           1200:
               gtyp_VGR.Workpiece.s_id := '0';
               gtyp_VGR.Workpiece.s_state := '';
               gtyp_VGR.Workpiece.s_type := '';
               FOR li_Counter := 1 TO 8 DO
                   gtyp_VGR.History[li_Counter].i_code := 0;
                   gtyp_VGR.History[li_Counter].ldt_ts := DT#1990-01-01-00:00:00.00;
               END_FOR;

               IF gtyp_HBW.x_HBW_Container_Available THEN
                   gtyp_VGR.x_HBW_Discards := TRUE;
               END_IF;

               IF gtyp_HBW.x_HBW_Discards_Accepted OR gtyp_HBW.x_HBW_PickedUp_Accepted THEN
                   gtyp_VGR.x_HBW_Discards := FALSE;
                   gtyp_VGR.x_HBW_PickedUp := FALSE;
                   gtyp_HBW.x_HBW_Discards_Accepted := FALSE;
                   gtyp_HBW.x_HBW_PickedUp_Accepted := FALSE;
               END_IF;

               li_Lights := 2;
               gtyp_VGR.vertical_Axis.x_Reference := TRUE;

               IF NOT gtyp_VGR.vertical_Axis.x_Referenced THEN
                   li_StepCase := 1210;
               END_IF;

           1210:
               IF gtyp_VGR.vertical_Axis.x_Referenced THEN
                   gtyp_VGR.vertical_Axis.x_Reference := FALSE;
                   li_StepCase := 1220;
               END_IF;

           1220:
               gtyp_VGR.horizontal_Axis.x_Reference := TRUE;

               IF NOT gtyp_VGR.horizontal_Axis.x_Referenced THEN
                   li_StepCase := 1230;
               END_IF;

           1230:
               IF gtyp_VGR.horizontal_Axis.x_Referenced THEN
                   gtyp_VGR.horizontal_Axis.x_Reference := FALSE;
                   li_StepCase := 1240;
               END_IF;

           1240:
               gtyp_VGR.rotate_Axis.x_Reference := TRUE;

               IF NOT gtyp_VGR.rotate_Axis.x_Referenced THEN
                   li_StepCase := 1250;
               END_IF;

           1250:
               IF gtyp_VGR.rotate_Axis.x_Referenced THEN
                   gtyp_VGR.rotate_Axis.x_Reference := FALSE;
                   li_StepCase := 1260;
               END_IF;

           1260:
               gtyp_VGR.horizontal_Axis.di_Target_Position := gtyp_VGR.di_Pos_NiO_horizontal;
               gtyp_VGR.horizontal_Axis.x_Start_Positioning := TRUE;
               gtyp_VGR.vertical_Axis.di_Target_Position := gtyp_VGR.di_Pos_NiO_vertical;
               gtyp_VGR.vertical_Axis.x_Start_Positioning := TRUE;
               gtyp_VGR.vertical_Axis.i_PWM := 500;
               gtyp_VGR.rotate_Axis.di_Target_Position := gtyp_VGR.di_Pos_NiO_rotate;
               gtyp_VGR.rotate_Axis.x_Start_Positioning := TRUE;

               IF (gtyp_VGR.horizontal_Axis.di_Actual_Position <= (gtyp_VGR.di_Pos_NiO_horizontal + gtyp_VGR.horizontal_Axis.Config.di_Pos_Window))
                   AND (gtyp_VGR.horizontal_Axis.di_Actual_Position >= (gtyp_VGR.di_Pos_NiO_horizontal - gtyp_VGR.horizontal_Axis.Config.di_Pos_Window))
                   AND gtyp_VGR.horizontal_Axis.x_Position_Reached THEN
                   gtyp_VGR.horizontal_Axis.x_Start_Positioning := FALSE;
               END_IF;

               IF (gtyp_VGR.vertical_Axis.di_Actual_Position <= (gtyp_VGR.di_Pos_NiO_vertical + gtyp_VGR.vertical_Axis.Config.di_Pos_Window))
                   AND (gtyp_VGR.vertical_Axis.di_Actual_Position >= (gtyp_VGR.di_Pos_NiO_vertical - gtyp_VGR.vertical_Axis.Config.di_Pos_Window))
                   AND gtyp_VGR.vertical_Axis.x_Position_Reached THEN
                   gtyp_VGR.vertical_Axis.x_Start_Positioning := FALSE;
               END_IF;

               IF (gtyp_VGR.rotate_Axis.di_Actual_Position <= (gtyp_VGR.di_Pos_NiO_rotate + gtyp_VGR.rotate_Axis.Config.di_Pos_Window))
                   AND (gtyp_VGR.rotate_Axis.di_Actual_Position >= (gtyp_VGR.di_Pos_NiO_rotate - gtyp_VGR.rotate_Axis.Config.di_Pos_Window))
                   AND gtyp_VGR.rotate_Axis.x_Position_Reached THEN
                   gtyp_VGR.rotate_Axis.x_Start_Positioning := FALSE;
               END_IF;

               IF (gtyp_VGR.horizontal_Axis.di_Actual_Position <= (gtyp_VGR.di_Pos_NiO_horizontal + gtyp_VGR.horizontal_Axis.Config.di_Pos_Window))
                   AND (gtyp_VGR.horizontal_Axis.di_Actual_Position >= (gtyp_VGR.di_Pos_NiO_horizontal - gtyp_VGR.horizontal_Axis.Config.di_Pos_Window))
                   AND gtyp_VGR.horizontal_Axis.x_Position_Reached
                   AND (gtyp_VGR.vertical_Axis.di_Actual_Position <= (gtyp_VGR.di_Pos_NiO_vertical + gtyp_VGR.vertical_Axis.Config.di_Pos_Window))
                   AND (gtyp_VGR.vertical_Axis.di_Actual_Position >= (gtyp_VGR.di_Pos_NiO_vertical - gtyp_VGR.vertical_Axis.Config.di_Pos_Window))
                   AND gtyp_VGR.vertical_Axis.x_Position_Reached
                   AND (gtyp_VGR.rotate_Axis.di_Actual_Position <= (gtyp_VGR.di_Pos_NiO_rotate + gtyp_VGR.rotate_Axis.Config.di_Pos_Window))
                   AND (gtyp_VGR.rotate_Axis.di_Actual_Position >= (gtyp_VGR.di_Pos_NiO_rotate - gtyp_VGR.rotate_Axis.Config.di_Pos_Window))
                   AND gtyp_VGR.rotate_Axis.x_Position_Reached THEN
                   gtyp_VGR.horizontal_Axis.x_Start_Positioning := FALSE;
                   gtyp_VGR.vertical_Axis.x_Start_Positioning := FALSE;
                   gtyp_VGR.rotate_Axis.x_Start_Positioning := FALSE;
                   gtyp_VGR.vertical_Axis.i_PWM := 800;
                   li_StepCase := 1270;
               END_IF;

           1270:
               QX_VGR_ValveVacuum_Q8 := FALSE;
               li_StepCase := 1280;

           1280:

               lx_Start_TON_Wait := TRUE;
               lt_TON_Wait := T#1000ms;

               IF lfb_TON_Wait.Q THEN
                   QX_VGR_Compressor_Q7  := FALSE;
                   lx_Start_TON_Wait               := FALSE;
                   gtyp_VGR.x_Workpiece_NiO := FALSE;
                   gtyp_VGR.x_HBW_Discards := FALSE;
                   li_Lights := 1;
                   li_StepCase            := 0;
               END_IF;

       ELSE
               ;
       END_CASE;

   ELSE
       gtyp_VGR.Workpiece.s_id := '';
       gtyp_VGR.Workpiece.s_state := '';
       gtyp_VGR.Workpiece.s_type := '';

       gtyp_VGR.x_State_Process := FALSE;
       gtyp_Interface_Dashboard.Subscribe.State_Order.ldt_ts := DT_TO_LDT(ldt_MQTT);
       gtyp_Interface_Dashboard.Subscribe.State_Order.s_state := 'WAITING_FOR_ORDER';
       gtyp_Interface_Dashboard.Subscribe.State_Order.s_type := '';
       FOR li_Counter := 1 TO 8 DO
           gtyp_VGR.History[li_Counter].i_code := 0;
           gtyp_VGR.History[li_Counter].ldt_ts := DT#1990-01-01-00:00:00.00;
       END_FOR;

       gtyp_VGR.x_Start_Park_Position    := FALSE;
       gtyp_VGR.x_Park_Position_Reached  := FALSE;
       gtyp_VGR.x_NFC_Start_First        := FALSE;
       gtyp_VGR.x_NFC_Start              := FALSE;
       gtyp_VGR.x_NFC_Completed          := FALSE;
       gtyp_VGR.x_HBW_Storage            := FALSE;
       gtyp_VGR.x_HBW_Outsource          := FALSE;
       gtyp_VGR.s_HBW_Outsource_Typ      := '';
       gtyp_VGR.x_HBW_Discards           := FALSE;
       gtyp_VGR.x_HBW_PickedUp           := FALSE;
       gtyp_VGR.x_MPO_Req_Discard        := FALSE;
       gtyp_VGR.x_MPO_Discards           := FALSE;
       gtyp_VGR.x_Ready_For_Outsource    := FALSE;
       gtyp_VGR.x_State_Process          := FALSE;
       gtyp_VGR.x_Workpiece_NiO          := FALSE;

       gtyp_VGR.vertical_Axis.i_PWM      := 800;

       li_Lights := 1;
       lx_Init := TRUE;
   END_IF;
END_FUNCTION_BLOCK

FUNCTION_BLOCK PRG_Order
   VAR
      lx_Init : Bool;
      li_StepCase : Int;
      lldt_ts_old : LDT;
      ldt_MQTT : Date_And_Time;
      li_Return_LDT : Int;
      lfb_TON_Wait : TON_TIME;
      lx_Start_TON_Wait : Bool;
   END_VAR

   IF lx_Init THEN
       lfb_TON_Wait(IN:= lx_Start_TON_Wait,PT:= T#20s);
       CASE li_StepCase OF

           0:
               lx_Start_TON_Wait := FALSE;
               li_StepCase := 10;

           10:
               IF (gtyp_Interface_Dashboard.Publish.OrderWorkpieceButton.ldt_ts > lldt_ts_old) THEN
                   li_Return_LDT := RD_SYS_T(ldt_MQTT);
                   gtyp_Interface_Dashboard.Subscribe.State_Order.ldt_ts := DT_TO_LDT(ldt_MQTT);
                   gtyp_Interface_Dashboard.Subscribe.State_Order.s_state := 'ORDERED';
                   gtyp_VGR.s_HBW_Outsource_Typ := gtyp_Interface_Dashboard.Publish.OrderWorkpieceButton.s_type;
                   gtyp_Interface_Dashboard.Subscribe.State_Order.s_type := gtyp_VGR.s_HBW_Outsource_Typ;
                   IF gtyp_VGR.x_Ready_For_Outsource THEN
                       lldt_ts_old := gtyp_Interface_Dashboard.Publish.OrderWorkpieceButton.ldt_ts;
                       gtyp_VGR.x_HBW_Outsource := TRUE;
                       li_StepCase := 20;
                   END_IF;
               END_IF;

           20:
               IF gtyp_VGR.x_HBW_PickedUp OR NOT gtyp_VGR.x_HBW_Outsource THEN
                   gtyp_VGR.x_HBW_Outsource := FALSE;
                   gtyp_VGR.s_HBW_Outsource_Typ := '';
                   li_StepCase := 0;
               END_IF;


       ELSE
                   ;
       END_CASE;

   ELSE
       lx_Init    := TRUE;
       lldt_ts_old:= DT#1970-01-01-00:00:00.00;
   END_IF;
END_FUNCTION_BLOCK

FUNCTION_BLOCK PRG_MPO_Set_Park_Position
   VAR
      lx_Init : Bool;
      lx_Start_TON_Wait : Bool;
      lt_TON_Wait : Time;
      li_StepCase : Int;
      lfb_TON_Wait : TON_TIME;
      lfb_R_Trig_Start_Park_Pos : R_TRIG;
   END_VAR



   IF lx_Init THEN


       lfb_TON_Wait(IN := lx_Start_TON_Wait,
                     PT := lt_TON_Wait);

       lfb_R_Trig_Start_Park_Pos(CLK := gtyp_Setup.x_Park_Position
                                  OR IX_Set_Park_Position);


       IF lfb_R_Trig_Start_Park_Pos.Q THEN
           gtyp_MPO.x_Start_Park_Position := TRUE;
           li_StepCase := 0;
       END_IF;


       IF NOT gtyp_MPO.x_Start_Park_Position THEN
           li_StepCase := 0;
       END_IF;


       CASE li_StepCase OF

           0:
               lx_Start_TON_Wait := FALSE;
               li_StepCase := 10;

           10:
               IF gtyp_MPO.x_Start_Park_Position AND NOT gtyp_MPO.x_Park_Position_Reached THEN
                   li_StepCase := 20;
               END_IF;

           20:
               QX_MPO_M5_VacuumTowardsTurnTable_Q8 := FALSE;
               QX_MPO_M5_VacuumTowardsOven_Q7    := TRUE;
               lx_Start_TON_Wait                  := TRUE;
               lt_TON_Wait                        := T#4000ms;

               IF lfb_TON_Wait.Q THEN
                   QX_MPO_M5_VacuumTowardsTurnTable_Q8 := FALSE;
                   QX_MPO_M5_VacuumTowardsOven_Q7    := FALSE;
                   lx_Start_TON_Wait                  := FALSE;
                   li_StepCase                        := 30;
               END_IF;

           30:
               QX_MPO_M1_TurnTableClockwise_Q1        := TRUE;
               QX_MPO_M1_TurnTableCounterclockwise_Q2 := FALSE;
               lx_Start_TON_Wait := TRUE;
               lt_TON_Wait := T#1000ms;

               IF lfb_TON_Wait.Q THEN
                   QX_MPO_M1_TurnTableClockwise_Q1 := FALSE;
                   QX_MPO_M1_TurnTableCounterclockwise_Q2 := FALSE;
                   lx_Start_TON_Wait := FALSE;
                   li_StepCase := 40;
               END_IF;

           40:
               gtyp_MPO.x_Park_Position_Reached := TRUE;



           ELSE
               ;
       END_CASE;

   ELSE
       lx_Init := TRUE;
   END_IF;
END_FUNCTION_BLOCK

FUNCTION_BLOCK PRG_HBW_Ablauf
   VAR
      lx_Init : Bool;
      lx_Start_TON_Fill_HBW : Bool;
      lx_Start_TON_Wait : Bool;
      lx_Time_Error : Bool;
      lt_TON_Wait : Time;
      lx_Start_TON_State : Bool;
      lx_Storage : Bool;
      ldt_MQTT : Date_And_Time;
      li_Return_LDT : Int;
      lldt_Outsource : LDT;
      li_Lights : Int;
      li_Lights_old : Int;
      li_Counter_Hor : Int;
      li_Counter_Ver : Int;
      li_Counter_Act_Hor : Int;
      li_Counter_Act_Ver : Int;
      li_Counter : Int;
      li_StepCase : Int;
      ldi_PosRack_Horizontal : DInt;
      ldi_PosRack_Vertical : DInt;
      ls_Color : String;
      lfb_TON_State : TON_TIME;
      lfb_TON_ConveyerBelt_Out : TON_TIME;
      lfb_TON_Wait : TON_TIME;
      lfb_TON_Fill_HBW : TON_TIME;
      lfb_TON_Error : TON_TIME;
   END_VAR

   IF lx_Init THEN
       IF gtyp_Setup.x_Set_Pos_Activ OR gtyp_HBW.x_Start_Park_Position THEN
           li_StepCase := 0;
       END_IF;


       lfb_TON_State(IN := NOT lx_Start_TON_State,
                       PT := T#2s);


       lfb_TON_Error(IN := lx_Time_Error,
                      PT := T#30s);


       lfb_TON_Fill_HBW(IN := lx_Start_TON_Fill_HBW,
                         PT := T#60s);

       IF lfb_TON_Fill_HBW.Q THEN
           lx_Start_TON_Fill_HBW:= FALSE;
       END_IF;

       IF lx_Start_TON_Fill_HBW AND (IX_Fill_HBW OR gtyp_Setup.x_Fill_Rack_HBW) THEN
           li_Return_LDT := RD_SYS_T(ldt_MQTT);

           gtyp_HBW.Rack_Workpiece[1, 1].s_id    := '04c34892186580';
           gtyp_HBW.Rack_Workpiece[1, 1].s_state := 'RAW';
           gtyp_HBW.Rack_Workpiece[1, 1].s_type  := 'WHITE';
           gtyp_HBW.Rack_History[1, 1].History[1].ldt_ts := DT_TO_LDT(ldt_MQTT);
           gtyp_HBW.Rack_History[1, 1].History[1].i_code := 100;
           gtyp_HBW.Rack_History[1, 1].History[2].ldt_ts := DT_TO_LDT(ldt_MQTT);
           gtyp_HBW.Rack_History[1, 1].History[2].i_code := 200;
           gtyp_HBW.Rack_History[1, 1].History[3].ldt_ts := DT_TO_LDT(ldt_MQTT);
           gtyp_HBW.Rack_History[1, 1].History[3].i_code := 300;

           gtyp_HBW.Rack_Workpiece[1, 2].s_id    := '04c34892186581';
           gtyp_HBW.Rack_Workpiece[1, 2].s_state := 'RAW';
           gtyp_HBW.Rack_Workpiece[1, 2].s_type  := 'WHITE';
           gtyp_HBW.Rack_History[1, 2].History[1].ldt_ts := DT_TO_LDT(ldt_MQTT);
           gtyp_HBW.Rack_History[1, 2].History[1].i_code := 100;
           gtyp_HBW.Rack_History[1, 2].History[2].ldt_ts := DT_TO_LDT(ldt_MQTT);
           gtyp_HBW.Rack_History[1, 2].History[2].i_code := 200;
           gtyp_HBW.Rack_History[1, 2].History[3].ldt_ts := DT_TO_LDT(ldt_MQTT);
           gtyp_HBW.Rack_History[1, 2].History[3].i_code := 300;

           gtyp_HBW.Rack_Workpiece[1, 3].s_id    := '04c34892186582';
           gtyp_HBW.Rack_Workpiece[1, 3].s_state := 'RAW';
           gtyp_HBW.Rack_Workpiece[1, 3].s_type  := 'WHITE';
           gtyp_HBW.Rack_History[1, 3].History[1].ldt_ts := DT_TO_LDT(ldt_MQTT);
           gtyp_HBW.Rack_History[1, 3].History[1].i_code := 100;
           gtyp_HBW.Rack_History[1, 3].History[2].ldt_ts := DT_TO_LDT(ldt_MQTT);
           gtyp_HBW.Rack_History[1, 3].History[2].i_code := 200;
           gtyp_HBW.Rack_History[1, 3].History[3].ldt_ts := DT_TO_LDT(ldt_MQTT);
           gtyp_HBW.Rack_History[1, 3].History[3].i_code := 300;

           gtyp_HBW.Rack_Workpiece[2, 1].s_id    := '04c34892186583';
           gtyp_HBW.Rack_Workpiece[2, 1].s_state := 'RAW';
           gtyp_HBW.Rack_Workpiece[2, 1].s_type  := 'RED';
           gtyp_HBW.Rack_History[2, 1].History[1].ldt_ts := DT_TO_LDT(ldt_MQTT);
           gtyp_HBW.Rack_History[2, 1].History[1].i_code := 100;
           gtyp_HBW.Rack_History[2, 1].History[2].ldt_ts := DT_TO_LDT(ldt_MQTT);
           gtyp_HBW.Rack_History[2, 1].History[2].i_code := 200;
           gtyp_HBW.Rack_History[2, 1].History[3].ldt_ts := DT_TO_LDT(ldt_MQTT);
           gtyp_HBW.Rack_History[2, 1].History[3].i_code := 300;

           gtyp_HBW.Rack_Workpiece[2, 2].s_id    := '04c34892186584';
           gtyp_HBW.Rack_Workpiece[2, 2].s_state := 'RAW';
           gtyp_HBW.Rack_Workpiece[2, 2].s_type  := 'RED';
           gtyp_HBW.Rack_History[2, 2].History[1].ldt_ts := DT_TO_LDT(ldt_MQTT);
           gtyp_HBW.Rack_History[2, 2].History[1].i_code := 100;
           gtyp_HBW.Rack_History[2, 2].History[2].ldt_ts := DT_TO_LDT(ldt_MQTT);
           gtyp_HBW.Rack_History[2, 2].History[2].i_code := 200;
           gtyp_HBW.Rack_History[2, 2].History[3].ldt_ts := DT_TO_LDT(ldt_MQTT);
           gtyp_HBW.Rack_History[2, 2].History[3].i_code := 300;

           gtyp_HBW.Rack_Workpiece[2, 3].s_id    := '04c34892186585';
           gtyp_HBW.Rack_Workpiece[2, 3].s_state := 'RAW';
           gtyp_HBW.Rack_Workpiece[2, 3].s_type  := 'RED';
           gtyp_HBW.Rack_History[2, 3].History[1].ldt_ts := DT_TO_LDT(ldt_MQTT);
           gtyp_HBW.Rack_History[2, 3].History[1].i_code := 100;
           gtyp_HBW.Rack_History[2, 3].History[2].ldt_ts := DT_TO_LDT(ldt_MQTT);
           gtyp_HBW.Rack_History[2, 3].History[2].i_code := 200;
           gtyp_HBW.Rack_History[2, 3].History[3].ldt_ts := DT_TO_LDT(ldt_MQTT);
           gtyp_HBW.Rack_History[2, 3].History[3].i_code := 300;

           gtyp_HBW.Rack_Workpiece[3, 1].s_id    := '04c34892186586';
           gtyp_HBW.Rack_Workpiece[3, 1].s_state := 'RAW';
           gtyp_HBW.Rack_Workpiece[3, 1].s_type  := 'BLUE';
           gtyp_HBW.Rack_History[3, 1].History[1].ldt_ts := DT_TO_LDT(ldt_MQTT);
           gtyp_HBW.Rack_History[3, 1].History[1].i_code := 100;
           gtyp_HBW.Rack_History[3, 1].History[2].ldt_ts := DT_TO_LDT(ldt_MQTT);
           gtyp_HBW.Rack_History[3, 1].History[2].i_code := 200;
           gtyp_HBW.Rack_History[3, 1].History[3].ldt_ts := DT_TO_LDT(ldt_MQTT);
           gtyp_HBW.Rack_History[3, 1].History[3].i_code := 300;

           gtyp_HBW.Rack_Workpiece[3, 2].s_id    := '04c34892186587';
           gtyp_HBW.Rack_Workpiece[3, 2].s_state := 'RAW';
           gtyp_HBW.Rack_Workpiece[3, 2].s_type  := 'BLUE';
           gtyp_HBW.Rack_History[3, 2].History[1].ldt_ts := DT_TO_LDT(ldt_MQTT);
           gtyp_HBW.Rack_History[3, 2].History[1].i_code := 100;
           gtyp_HBW.Rack_History[3, 2].History[2].ldt_ts := DT_TO_LDT(ldt_MQTT);
           gtyp_HBW.Rack_History[3, 2].History[2].i_code := 200;
           gtyp_HBW.Rack_History[3, 2].History[3].ldt_ts := DT_TO_LDT(ldt_MQTT);
           gtyp_HBW.Rack_History[3, 2].History[3].i_code := 300;

           gtyp_HBW.Rack_Workpiece[3, 3].s_id    := '04c34892186588';
           gtyp_HBW.Rack_Workpiece[3, 3].s_state := 'RAW';
           gtyp_HBW.Rack_Workpiece[3, 3].s_type  := 'BLUE';
           gtyp_HBW.Rack_History[3, 3].History[1].ldt_ts := DT_TO_LDT(ldt_MQTT);
           gtyp_HBW.Rack_History[3, 3].History[1].i_code := 100;
           gtyp_HBW.Rack_History[3, 3].History[2].ldt_ts := DT_TO_LDT(ldt_MQTT);
           gtyp_HBW.Rack_History[3, 3].History[2].i_code := 200;
           gtyp_HBW.Rack_History[3, 3].History[3].ldt_ts := DT_TO_LDT(ldt_MQTT);
           gtyp_HBW.Rack_History[3, 3].History[3].i_code := 300;

           lx_Start_TON_Fill_HBW          := FALSE;
           gtyp_Setup.x_Fill_Rack_HBW    := FALSE;
       END_IF;

       gtyp_Setup.x_Start_TON_Fill_HBW := lx_Start_TON_Fill_HBW;


        IF (lfb_TON_State.Q OR (li_Lights <> li_Lights_old)) AND NOT lx_Start_TON_State THEN
           li_Lights_old := li_Lights;
           lx_Start_TON_State := TRUE;
           li_Return_LDT := RD_SYS_T(ldt_MQTT);
           gtyp_Interface_Dashboard.Subscribe.Stock_HBW.StockItem := gtyp_HBW.Rack_Workpiece;
           gtyp_Interface_Dashboard.Subscribe.Stock_HBW.ldt_ts := DT_TO_LDT(ldt_MQTT);

           gtyp_Interface_Dashboard.Subscribe.State_HBW.ldt_ts := DT_TO_LDT(ldt_MQTT);
           gtyp_Interface_Dashboard.Subscribe.State_HBW.i_code := li_Lights;
           gtyp_Interface_Dashboard.Subscribe.State_HBW.s_description := '';
           gtyp_Interface_Dashboard.Subscribe.State_HBW.s_station := 'hbw';
           gtyp_Interface_Dashboard.Subscribe.State_HBW.s_target := '';
       END_IF;


       IF NOT lfb_TON_State.Q AND lx_Start_TON_State THEN
           lx_Start_TON_State := FALSE;
       END_IF;


       lfb_TON_Wait(IN := lx_Start_TON_Wait,
                       PT := lt_TON_Wait);


       lfb_TON_ConveyerBelt_Out(IN := NOT IX_HBW_LightBarrierOutside_I3,
                                 PT := T#300ms);



       gtyp_HBW.Rack_Pos[1, 1].di_PosRack_Horizontal := gtyp_HBW.di_PosRack_A1_Horizontal;
       gtyp_HBW.Rack_Pos[2, 1].di_PosRack_Horizontal := gtyp_HBW.di_PosRack_A1_Horizontal;
       gtyp_HBW.Rack_Pos[3, 1].di_PosRack_Horizontal := gtyp_HBW.di_PosRack_A1_Horizontal;

       gtyp_HBW.Rack_Pos[1, 2].di_PosRack_Horizontal := gtyp_HBW.di_PosRack_B2_Horizontal;
       gtyp_HBW.Rack_Pos[2, 2].di_PosRack_Horizontal := gtyp_HBW.di_PosRack_B2_Horizontal;
       gtyp_HBW.Rack_Pos[3, 2].di_PosRack_Horizontal := gtyp_HBW.di_PosRack_B2_Horizontal;

       gtyp_HBW.Rack_Pos[1, 3].di_PosRack_Horizontal := gtyp_HBW.di_PosRack_C3_Horizontal;
       gtyp_HBW.Rack_Pos[2, 3].di_PosRack_Horizontal := gtyp_HBW.di_PosRack_C3_Horizontal;
       gtyp_HBW.Rack_Pos[3, 3].di_PosRack_Horizontal := gtyp_HBW.di_PosRack_C3_Horizontal;

       gtyp_HBW.Rack_Pos[1, 1].di_PosRack_Vertical := gtyp_HBW.di_PosRack_A1_Vertical;
       gtyp_HBW.Rack_Pos[1, 2].di_PosRack_Vertical := gtyp_HBW.di_PosRack_A1_Vertical;
       gtyp_HBW.Rack_Pos[1, 3].di_PosRack_Vertical := gtyp_HBW.di_PosRack_A1_Vertical;

       gtyp_HBW.Rack_Pos[2, 1].di_PosRack_Vertical := gtyp_HBW.di_PosRack_B2_Vertical;
       gtyp_HBW.Rack_Pos[2, 2].di_PosRack_Vertical := gtyp_HBW.di_PosRack_B2_Vertical;
       gtyp_HBW.Rack_Pos[2, 3].di_PosRack_Vertical := gtyp_HBW.di_PosRack_B2_Vertical;

       gtyp_HBW.Rack_Pos[3, 1].di_PosRack_Vertical := gtyp_HBW.di_PosRack_C3_Vertical;
       gtyp_HBW.Rack_Pos[3, 2].di_PosRack_Vertical := gtyp_HBW.di_PosRack_C3_Vertical;
       gtyp_HBW.Rack_Pos[3, 3].di_PosRack_Vertical := gtyp_HBW.di_PosRack_C3_Vertical;


       CASE li_StepCase OF

           0:
               lx_Start_TON_Wait := FALSE;
               lx_Time_Error := FALSE;

               gtyp_HBW.Horizontal_Axis.x_Start_Positioning := FALSE;
               gtyp_HBW.Vertical_Axis.x_Start_Positioning := FALSE;
               gtyp_HBW.Horizontal_Axis.x_Reference := FALSE;
               gtyp_HBW.Vertical_Axis.x_Reference := FALSE;

               IF NOT gtyp_HBW.x_Error AND NOT gtyp_Setup.x_Set_Pos_Activ AND NOT gtyp_HBW.x_Start_Park_Position THEN
                   li_StepCase := 10;
               END_IF;

           10:
               li_Lights := 2;
               IF IX_HBW_SwitchCantileverFront_I5 OR NOT IX_HBW_SwitchCantileverBack_I6 THEN
                   QX_HBW_M4_CantileverBackward_Q8 := TRUE;
                   QX_HBW_M4_CantileverForward_Q7 := FALSE;
               ELSIF NOT IX_HBW_SwitchCantileverFront_I5 AND IX_HBW_SwitchCantileverBack_I6 THEN
                   QX_HBW_M4_CantileverBackward_Q8 := FALSE;
                   QX_HBW_M4_CantileverForward_Q7 := FALSE;
                   li_StepCase := 20;
               END_IF;

           20:

               gtyp_HBW.Horizontal_Axis.x_Reference := TRUE;
               gtyp_HBW.Vertical_Axis.x_Reference := TRUE;

               IF NOT gtyp_HBW.Horizontal_Axis.x_Referenced AND NOT gtyp_HBW.Vertical_Axis.x_Referenced THEN
                   li_StepCase := 30;
               END_IF;

           30:
               IF gtyp_HBW.Horizontal_Axis.x_Referenced THEN
                   gtyp_HBW.Horizontal_Axis.x_Reference := FALSE;
               END_IF;
               IF gtyp_HBW.Vertical_Axis.x_Referenced THEN
                   gtyp_HBW.Vertical_Axis.x_Reference := FALSE;
               END_IF;

               IF gtyp_HBW.Horizontal_Axis.x_Referenced AND gtyp_HBW.Vertical_Axis.x_Referenced THEN
                   gtyp_HBW.Horizontal_Axis.x_Reference := FALSE;
                   gtyp_HBW.Vertical_Axis.x_Reference := FALSE;
                   li_StepCase := 40;
               END_IF;

           40:

               li_Lights := 1;
               lx_Storage := FALSE;


               IF gtyp_VGR.x_HBW_Storage THEN
                   li_Lights := 2;
                   li_StepCase := 50;

               ELSIF gtyp_VGR.x_HBW_Outsource THEN
                   li_Lights := 2;
                   li_StepCase := 60;
               END_IF;

           50:
               FOR li_Counter_Hor := 1 TO 3 DO
                   FOR li_Counter_Ver := 1 TO 3 DO
                       IF gtyp_HBW.Rack_Workpiece[li_Counter_Ver, li_Counter_Hor].s_id = '0' THEN
                           li_Counter_Act_Hor := li_Counter_Hor;
                           li_Counter_Act_Ver := li_Counter_Ver;
                           ldi_PosRack_Horizontal := gtyp_HBW.Rack_Pos[li_Counter_Ver, li_Counter_Hor].di_PosRack_Horizontal;
                           ldi_PosRack_Vertical := gtyp_HBW.Rack_Pos[li_Counter_Ver, li_Counter_Hor].di_PosRack_Vertical;
                           li_StepCase := 70;
                       END_IF;
                       IF li_StepCase = 70 THEN
                           EXIT;
                       END_IF;
                   END_FOR;
                   IF li_StepCase = 70 THEN
                       EXIT;
                   END_IF;
               END_FOR;

           60:
               li_Return_LDT := RD_SYS_T(ldt_MQTT);
               lldt_Outsource := ldt_MQTT;

               FOR li_Counter_Hor := 1 TO 3 DO
                   FOR li_Counter_Ver := 1 TO 3 DO
                       IF (gtyp_VGR.s_HBW_Outsource_Typ = gtyp_HBW.Rack_Workpiece[li_Counter_Ver, li_Counter_Hor].s_type)
                           AND (lldt_Outsource > gtyp_HBW.Rack_History[li_Counter_Ver, li_Counter_Hor].History[3].ldt_ts)
                           AND NOT (gtyp_HBW.Rack_History[li_Counter_Ver, li_Counter_Hor].History[3].ldt_ts = DT#1970-01-01-00:00:00.00) THEN
                           lldt_Outsource := gtyp_HBW.Rack_History[li_Counter_Ver, li_Counter_Hor].History[3].ldt_ts;
                           li_Counter_Act_Hor := li_Counter_Hor;
                           li_Counter_Act_Ver := li_Counter_Ver;
                           ldi_PosRack_Horizontal := gtyp_HBW.Rack_Pos[li_Counter_Ver, li_Counter_Hor].di_PosRack_Horizontal;
                           ldi_PosRack_Vertical := gtyp_HBW.Rack_Pos[li_Counter_Ver, li_Counter_Hor].di_PosRack_Vertical;
                       END_IF;
                   END_FOR;
               END_FOR;

               IF (li_Counter_Act_Hor = 4) OR (li_Counter_Act_Ver = 4) THEN
                   li_StepCase := 40;
               ELSE
                   li_StepCase := 70;
               END_IF;

           70:
               gtyp_HBW.Horizontal_Axis.di_Target_Position := ldi_PosRack_Horizontal;
               gtyp_HBW.Horizontal_Axis.x_Start_Positioning := TRUE;
               gtyp_HBW.Vertical_Axis.di_Target_Position := ldi_PosRack_Vertical;
               gtyp_HBW.Vertical_Axis.x_Start_Positioning := TRUE;

               IF (gtyp_HBW.Horizontal_Axis.di_Actual_Position <= (ldi_PosRack_Horizontal + gtyp_HBW.Horizontal_Axis.Config.di_Pos_Window))
                   AND (gtyp_HBW.Horizontal_Axis.di_Actual_Position >= (ldi_PosRack_Horizontal - gtyp_HBW.Horizontal_Axis.Config.di_Pos_Window))
                   AND gtyp_HBW.Horizontal_Axis.x_Position_Reached THEN
                   gtyp_HBW.Horizontal_Axis.x_Start_Positioning := FALSE;
               END_IF;

               IF (gtyp_HBW.Vertical_Axis.di_Actual_Position <= (ldi_PosRack_Vertical + gtyp_HBW.Vertical_Axis.Config.di_Pos_Window))
                   AND (gtyp_HBW.Vertical_Axis.di_Actual_Position >= (ldi_PosRack_Vertical - gtyp_HBW.Vertical_Axis.Config.di_Pos_Window))
                   AND gtyp_HBW.Vertical_Axis.x_Position_Reached THEN
                   gtyp_HBW.Vertical_Axis.x_Start_Positioning := FALSE;
               END_IF;

               IF (gtyp_HBW.Horizontal_Axis.di_Actual_Position <= (ldi_PosRack_Horizontal + gtyp_HBW.Horizontal_Axis.Config.di_Pos_Window))
                   AND (gtyp_HBW.Horizontal_Axis.di_Actual_Position >= (ldi_PosRack_Horizontal - gtyp_HBW.Horizontal_Axis.Config.di_Pos_Window))
                   AND gtyp_HBW.Horizontal_Axis.x_Position_Reached
                   AND (gtyp_HBW.Vertical_Axis.di_Actual_Position <= (ldi_PosRack_Vertical + gtyp_HBW.Vertical_Axis.Config.di_Pos_Window))
                   AND (gtyp_HBW.Vertical_Axis.di_Actual_Position >= (ldi_PosRack_Vertical - gtyp_HBW.Vertical_Axis.Config.di_Pos_Window))
                   AND gtyp_HBW.Vertical_Axis.x_Position_Reached THEN
                   gtyp_HBW.Horizontal_Axis.x_Start_Positioning := FALSE;
                   gtyp_HBW.Vertical_Axis.x_Start_Positioning := FALSE;
                   li_StepCase := 80;
               END_IF;

           80:

               QX_HBW_M4_CantileverBackward_Q8 := FALSE;
               QX_HBW_M4_CantileverForward_Q7 := TRUE;

               IF IX_HBW_SwitchCantileverFront_I5 AND NOT IX_HBW_SwitchCantileverBack_I6 THEN
                   QX_HBW_M4_CantileverBackward_Q8 := FALSE;
                   QX_HBW_M4_CantileverForward_Q7 := FALSE;
                   li_StepCase := 90;
               END_IF;

           90:
               gtyp_HBW.Vertical_Axis.di_Target_Position := ldi_PosRack_Vertical - gtyp_HBW.di_Offset_Pos_Rack_Vertical;
               gtyp_HBW.Vertical_Axis.x_Start_Positioning := TRUE;

               IF (gtyp_HBW.Vertical_Axis.di_Actual_Position <= (ldi_PosRack_Vertical - gtyp_HBW.di_Offset_Pos_Rack_Vertical + gtyp_HBW.Vertical_Axis.Config.di_Pos_Window))
                   AND (gtyp_HBW.Vertical_Axis.di_Actual_Position >= (ldi_PosRack_Vertical - gtyp_HBW.di_Offset_Pos_Rack_Vertical - gtyp_HBW.Vertical_Axis.Config.di_Pos_Window))
                   AND gtyp_HBW.Vertical_Axis.x_Position_Reached THEN
                   gtyp_HBW.Vertical_Axis.x_Start_Positioning := FALSE;
                   li_StepCase := 100;
               END_IF;

           100:

               QX_HBW_M4_CantileverBackward_Q8 := TRUE;
               QX_HBW_M4_CantileverForward_Q7 := FALSE;

               IF NOT IX_HBW_SwitchCantileverFront_I5 AND IX_HBW_SwitchCantileverBack_I6 THEN
                   IF gtyp_VGR.x_HBW_Storage THEN
                       gtyp_HBW.Rack_Workpiece[li_Counter_Act_Ver, li_Counter_Act_Hor].s_id := '';
                   ELSIF gtyp_VGR.x_HBW_Outsource THEN
                       gtyp_Interface_Dashboard.Subscribe.State_HBW.x_active := TRUE;
                       gtyp_HBW.History := gtyp_HBW.Rack_History[li_Counter_Act_Ver, li_Counter_Act_Hor].History;
                       gtyp_HBW.Workpiece := gtyp_HBW.Rack_Workpiece[li_Counter_Act_Ver, li_Counter_Act_Hor];
                       li_Return_LDT := RD_SYS_T(ldt_MQTT);
                       gtyp_HBW.History[4].i_code := 400;
                       gtyp_HBW.History[4].ldt_ts := DT_TO_LDT(ldt_MQTT);

                       gtyp_HBW.Rack_Workpiece[li_Counter_Act_Ver, li_Counter_Act_Hor].s_id := '';
                       gtyp_HBW.Rack_Workpiece[li_Counter_Act_Ver, li_Counter_Act_Hor].s_state := '';
                       gtyp_HBW.Rack_Workpiece[li_Counter_Act_Ver, li_Counter_Act_Hor].s_type := '';
                       FOR li_Counter := 1 TO 8 DO
                           gtyp_HBW.Rack_History[li_Counter_Act_Ver, li_Counter_Act_Hor].History[li_Counter].i_code := 0;
                           gtyp_HBW.Rack_History[li_Counter_Act_Ver, li_Counter_Act_Hor].History[li_Counter].ldt_ts := DT#1990-01-01-00:00:00.00;
                       END_FOR;
                   END_IF;
                   QX_HBW_M4_CantileverBackward_Q8 := FALSE;
                   QX_HBW_M4_CantileverForward_Q7 := FALSE;
                   li_StepCase := 110;
               END_IF;

           110:

               gtyp_HBW.Horizontal_Axis.x_Reference := TRUE;

               gtyp_HBW.Vertical_Axis.di_Target_Position := gtyp_HBW.di_PosBelt_Vertical - gtyp_HBW.di_Offset_Pos_Belt_Vertical;
               gtyp_HBW.Vertical_Axis.x_Start_Positioning := TRUE;

               IF (gtyp_HBW.Vertical_Axis.di_Actual_Position <= (gtyp_HBW.di_PosBelt_Vertical - gtyp_HBW.di_Offset_Pos_Belt_Vertical + gtyp_HBW.Vertical_Axis.Config.di_Pos_Window))
                   AND (gtyp_HBW.Vertical_Axis.di_Actual_Position >= (gtyp_HBW.di_PosBelt_Vertical - gtyp_HBW.di_Offset_Pos_Belt_Vertical - gtyp_HBW.Vertical_Axis.Config.di_Pos_Window))
                   AND gtyp_HBW.Vertical_Axis.x_Position_Reached THEN
                   gtyp_HBW.Vertical_Axis.x_Start_Positioning := FALSE;
               END_IF;

               IF NOT gtyp_HBW.Horizontal_Axis.x_Referenced THEN
                   li_StepCase := 120;
               END_IF;

           120:

               IF gtyp_HBW.Horizontal_Axis.x_Referenced THEN
                   gtyp_HBW.Horizontal_Axis.x_Reference := FALSE;
               END_IF;

               IF (gtyp_HBW.Vertical_Axis.di_Actual_Position <= (gtyp_HBW.di_PosBelt_Vertical - gtyp_HBW.di_Offset_Pos_Belt_Vertical + gtyp_HBW.Vertical_Axis.Config.di_Pos_Window))
                   AND (gtyp_HBW.Vertical_Axis.di_Actual_Position >= (gtyp_HBW.di_PosBelt_Vertical - gtyp_HBW.di_Offset_Pos_Belt_Vertical - gtyp_HBW.Vertical_Axis.Config.di_Pos_Window))
                   AND gtyp_HBW.Vertical_Axis.x_Position_Reached THEN
                   gtyp_HBW.Vertical_Axis.x_Start_Positioning := FALSE;
               END_IF;

               IF gtyp_HBW.Horizontal_Axis.x_Referenced
                   AND (gtyp_HBW.Vertical_Axis.di_Actual_Position <= (gtyp_HBW.di_PosBelt_Vertical - gtyp_HBW.di_Offset_Pos_Belt_Vertical + gtyp_HBW.Vertical_Axis.Config.di_Pos_Window))
                   AND (gtyp_HBW.Vertical_Axis.di_Actual_Position >= (gtyp_HBW.di_PosBelt_Vertical - gtyp_HBW.di_Offset_Pos_Belt_Vertical - gtyp_HBW.Vertical_Axis.Config.di_Pos_Window))
                   AND gtyp_HBW.Vertical_Axis.x_Position_Reached  THEN
                   gtyp_HBW.Horizontal_Axis.x_Reference := FALSE;
                   gtyp_HBW.Vertical_Axis.x_Start_Positioning := FALSE;
                   li_StepCase := 130;
               END_IF;

           130:
               gtyp_HBW.Horizontal_Axis.di_Target_Position := gtyp_HBW.di_PosBelt_Horizontal;
               gtyp_HBW.Horizontal_Axis.x_Start_Positioning := TRUE;

               IF (gtyp_HBW.Horizontal_Axis.di_Actual_Position <= (gtyp_HBW.di_PosBelt_Horizontal + gtyp_HBW.Horizontal_Axis.Config.di_Pos_Window))
                   AND (gtyp_HBW.Horizontal_Axis.di_Actual_Position >= (gtyp_HBW.di_PosBelt_Horizontal - gtyp_HBW.Horizontal_Axis.Config.di_Pos_Window))
                   AND gtyp_HBW.Horizontal_Axis.x_Position_Reached THEN
                   gtyp_HBW.Horizontal_Axis.x_Start_Positioning := FALSE;
               END_IF;

               IF (gtyp_HBW.Horizontal_Axis.di_Actual_Position <= (gtyp_HBW.di_PosBelt_Horizontal + gtyp_HBW.Horizontal_Axis.Config.di_Pos_Window))
                   AND (gtyp_HBW.Horizontal_Axis.di_Actual_Position >= (gtyp_HBW.di_PosBelt_Horizontal - gtyp_HBW.Horizontal_Axis.Config.di_Pos_Window))
                   AND gtyp_HBW.Horizontal_Axis.x_Position_Reached THEN
                   gtyp_HBW.Horizontal_Axis.x_Start_Positioning := FALSE;
                   li_StepCase := 140;
               END_IF;

           140:

               QX_HBW_M4_CantileverBackward_Q8 := FALSE;
               QX_HBW_M4_CantileverForward_Q7 := TRUE;

               lx_Time_Error := TRUE;

               IF IX_HBW_SwitchCantileverFront_I5 AND NOT IX_HBW_SwitchCantileverBack_I6 THEN
                   QX_HBW_M4_CantileverBackward_Q8   := FALSE;
                   QX_HBW_M4_CantileverForward_Q7    := FALSE;
                   lx_Time_Error                      := FALSE;
                   li_StepCase := 150;
               END_IF;


               IF lfb_TON_Error.Q THEN
                   li_Lights := 4;
                   lx_Time_Error := FALSE;
                   QX_HBW_M1_ConveyorBeltBackward_Q2 := FALSE;
                   QX_HBW_M1_ConveyorBeltForward_Q1 := FALSE;
                   gtyp_Interface_Dashboard.Subscribe.State_HBW.x_active := FALSE;
                   gtyp_HBW.x_Error := TRUE;
                   li_StepCase := 0;
               END_IF;

           150:
               gtyp_HBW.Vertical_Axis.di_Target_Position := gtyp_HBW.di_PosBelt_Vertical;
               gtyp_HBW.Vertical_Axis.x_Start_Positioning := TRUE;

               IF (gtyp_HBW.Vertical_Axis.di_Actual_Position <= (gtyp_HBW.di_PosBelt_Vertical + gtyp_HBW.Vertical_Axis.Config.di_Pos_Window))
                   AND (gtyp_HBW.Vertical_Axis.di_Actual_Position >= (gtyp_HBW.di_PosBelt_Vertical - gtyp_HBW.Vertical_Axis.Config.di_Pos_Window))
                   AND gtyp_HBW.Vertical_Axis.x_Position_Reached THEN
                   gtyp_HBW.Vertical_Axis.x_Start_Positioning := FALSE;
                   li_StepCase := 160;
               END_IF;

           160:

               lx_Time_Error := TRUE;

               IF NOT IX_HBW_LightBarrierInside_I2 THEN
                   QX_HBW_M1_ConveyorBeltBackward_Q2 := FALSE;
                   QX_HBW_M1_ConveyorBeltForward_Q1  := TRUE;
                   lx_Time_Error                      := FALSE;
                   li_StepCase                        := 170;
               END_IF;


               IF lfb_TON_Error.Q THEN
                   li_Lights := 4;
                   lx_Time_Error := FALSE;
                   QX_HBW_M1_ConveyorBeltBackward_Q2 := FALSE;
                   QX_HBW_M1_ConveyorBeltForward_Q1 := FALSE;
                   gtyp_Interface_Dashboard.Subscribe.State_HBW.x_active := FALSE;
                   gtyp_HBW.x_Error := TRUE;
                   li_StepCase := 0;
               END_IF;

           170:

               lx_Time_Error := TRUE;

               IF lfb_TON_ConveyerBelt_Out.Q THEN
                   QX_HBW_M1_ConveyorBeltBackward_Q2 := FALSE;
                   QX_HBW_M1_ConveyorBeltForward_Q1 := FALSE;
                   gtyp_HBW.x_HBW_Container_Available := TRUE;
                   lx_Time_Error := FALSE;
                   li_StepCase := 180;
               END_IF;


               IF lfb_TON_Error.Q THEN
                   li_Lights := 4;
                   lx_Time_Error := FALSE;
                   QX_HBW_M1_ConveyorBeltBackward_Q2 := FALSE;
                   QX_HBW_M1_ConveyorBeltForward_Q1 := FALSE;
                   gtyp_Interface_Dashboard.Subscribe.State_HBW.x_active := FALSE;
                   gtyp_HBW.x_Error := TRUE;
                   li_StepCase := 0;
               END_IF;

           180:

               li_Lights := 1;

               IF gtyp_VGR.x_HBW_PickedUp AND gtyp_VGR.x_HBW_Outsource THEN
                   gtyp_VGR.Workpiece := gtyp_HBW.Workpiece;
                   gtyp_VGR.History   := gtyp_HBW.History;
                   gtyp_HBW.Workpiece.s_id := '0';
                   gtyp_HBW.Workpiece.s_state := '';
                   gtyp_HBW.Workpiece.s_type := '';
                   FOR li_Counter := 1 TO 8 DO
                       gtyp_HBW.History[li_Counter].i_code := 0;
                       gtyp_HBW.History[li_Counter].ldt_ts := DT#1990-01-01-00:00:00.00;
                   END_FOR;
                   gtyp_HBW.x_HBW_Container_Available := FALSE;
                   gtyp_HBW.x_HBW_PickedUp_Accepted := TRUE;

                   gtyp_Interface_Dashboard.Subscribe.State_HBW.x_active := FALSE;

                   li_Lights := 2;
                   li_StepCase := 190;

               ELSIF gtyp_VGR.x_HBW_Discards AND gtyp_VGR.x_HBW_Storage THEN
                   gtyp_Interface_Dashboard.Subscribe.State_HBW.x_active := TRUE;
                   gtyp_HBW.Workpiece := gtyp_VGR.Workpiece;
                   gtyp_HBW.History:= gtyp_VGR.History;
                   gtyp_HBW.x_HBW_Container_Available := FALSE;
                   gtyp_HBW.x_HBW_Discards_Accepted := TRUE;
                   lx_Storage := true;

                   li_Lights := 2;
                   li_StepCase := 190;
               END_IF;

           190:

               IF NOT gtyp_VGR.x_HBW_Discards AND NOT gtyp_VGR.x_HBW_PickedUp THEN
                   QX_HBW_M1_ConveyorBeltBackward_Q2 := TRUE;
                   QX_HBW_M1_ConveyorBeltForward_Q1 := FALSE;
                   li_StepCase := 200;
               END_IF;

           200:

               lx_Time_Error := TRUE;

               IF NOT IX_HBW_LightBarrierInside_I2 THEN
                   QX_HBW_M1_ConveyorBeltBackward_Q2 := FALSE;
                   QX_HBW_M1_ConveyorBeltForward_Q1  := FALSE;
                   lx_Time_Error                      := FALSE;
                   li_StepCase                        := 210;
               END_IF;


               IF lfb_TON_Error.Q THEN
                   li_Lights := 4;
                   lx_Time_Error := FALSE;
                   QX_HBW_M1_ConveyorBeltBackward_Q2 := FALSE;
                   QX_HBW_M1_ConveyorBeltForward_Q1 := FALSE;
                   gtyp_Interface_Dashboard.Subscribe.State_HBW.x_active := FALSE;
                   gtyp_HBW.x_Error := TRUE;
                   li_StepCase := 0;
               END_IF;

           210:

               gtyp_HBW.Vertical_Axis.di_Target_Position := gtyp_HBW.di_PosBelt_Vertical - gtyp_HBW.di_Offset_Pos_Belt_Vertical;
               gtyp_HBW.Vertical_Axis.x_Start_Positioning := TRUE;

               IF (gtyp_HBW.Vertical_Axis.di_Actual_Position <= (gtyp_HBW.di_PosBelt_Vertical - gtyp_HBW.di_Offset_Pos_Belt_Vertical + gtyp_HBW.Vertical_Axis.Config.di_Pos_Window))
                   AND (gtyp_HBW.Vertical_Axis.di_Actual_Position >= (gtyp_HBW.di_PosBelt_Vertical - gtyp_HBW.di_Offset_Pos_Belt_Vertical - gtyp_HBW.Vertical_Axis.Config.di_Pos_Window))
                   AND gtyp_HBW.Vertical_Axis.x_Position_Reached THEN
                   gtyp_HBW.Vertical_Axis.x_Start_Positioning := FALSE;
               END_IF;

               IF (gtyp_HBW.Vertical_Axis.di_Actual_Position <= (gtyp_HBW.di_PosBelt_Vertical - gtyp_HBW.di_Offset_Pos_Belt_Vertical + gtyp_HBW.Vertical_Axis.Config.di_Pos_Window))
                   AND (gtyp_HBW.Vertical_Axis.di_Actual_Position >= (gtyp_HBW.di_PosBelt_Vertical - gtyp_HBW.di_Offset_Pos_Belt_Vertical - gtyp_HBW.Vertical_Axis.Config.di_Pos_Window))
                   AND gtyp_HBW.Vertical_Axis.x_Position_Reached THEN
                   gtyp_HBW.Vertical_Axis.x_Start_Positioning := FALSE;
                   li_StepCase := 220;
               END_IF;

           220:
               QX_HBW_M4_CantileverBackward_Q8 := TRUE;
               QX_HBW_M4_CantileverForward_Q7 := FALSE;

               IF NOT IX_HBW_SwitchCantileverFront_I5 AND IX_HBW_SwitchCantileverBack_I6 THEN
                   QX_HBW_M4_CantileverBackward_Q8 := FALSE;
                   QX_HBW_M4_CantileverForward_Q7 := FALSE;
                   li_StepCase := 230;
               END_IF;

           230:
               gtyp_HBW.Horizontal_Axis.di_Target_Position := ldi_PosRack_Horizontal;
               gtyp_HBW.Horizontal_Axis.x_Start_Positioning := TRUE;
               gtyp_HBW.Vertical_Axis.di_Target_Position := ldi_PosRack_Vertical - gtyp_HBW.di_Offset_Pos_Rack_Vertical;
               gtyp_HBW.Vertical_Axis.x_Start_Positioning := TRUE;

               IF (gtyp_HBW.Horizontal_Axis.di_Actual_Position <= (ldi_PosRack_Horizontal + gtyp_HBW.Horizontal_Axis.Config.di_Pos_Window))
                   AND (gtyp_HBW.Horizontal_Axis.di_Actual_Position >= (ldi_PosRack_Horizontal - gtyp_HBW.Horizontal_Axis.Config.di_Pos_Window))
                   AND gtyp_HBW.Horizontal_Axis.x_Position_Reached THEN
                   gtyp_HBW.Horizontal_Axis.x_Start_Positioning := FALSE;
               END_IF;

               IF (gtyp_HBW.Vertical_Axis.di_Actual_Position <= (ldi_PosRack_Vertical - gtyp_HBW.di_Offset_Pos_Rack_Vertical + gtyp_HBW.Vertical_Axis.Config.di_Pos_Window))
                   AND (gtyp_HBW.Vertical_Axis.di_Actual_Position >= (ldi_PosRack_Vertical - gtyp_HBW.di_Offset_Pos_Rack_Vertical - gtyp_HBW.Vertical_Axis.Config.di_Pos_Window))
                   AND gtyp_HBW.Vertical_Axis.x_Position_Reached THEN
                   gtyp_HBW.Vertical_Axis.x_Start_Positioning := FALSE;
               END_IF;

               IF (gtyp_HBW.Horizontal_Axis.di_Actual_Position <= (ldi_PosRack_Horizontal + gtyp_HBW.Horizontal_Axis.Config.di_Pos_Window))
                   AND (gtyp_HBW.Horizontal_Axis.di_Actual_Position >= (ldi_PosRack_Horizontal - gtyp_HBW.Horizontal_Axis.Config.di_Pos_Window))
                   AND gtyp_HBW.Horizontal_Axis.x_Position_Reached
                   AND (gtyp_HBW.Vertical_Axis.di_Actual_Position <= (ldi_PosRack_Vertical - gtyp_HBW.di_Offset_Pos_Rack_Vertical + gtyp_HBW.Vertical_Axis.Config.di_Pos_Window))
                   AND (gtyp_HBW.Vertical_Axis.di_Actual_Position >= (ldi_PosRack_Vertical - gtyp_HBW.di_Offset_Pos_Rack_Vertical - gtyp_HBW.Vertical_Axis.Config.di_Pos_Window))
                   AND gtyp_HBW.Vertical_Axis.x_Position_Reached THEN
                   gtyp_HBW.Horizontal_Axis.x_Start_Positioning := FALSE;
                   gtyp_HBW.Vertical_Axis.x_Start_Positioning := FALSE;
                   li_StepCase := 240;
               END_IF;

           240:

               QX_HBW_M4_CantileverBackward_Q8 := FALSE;
               QX_HBW_M4_CantileverForward_Q7 := TRUE;

               IF IX_HBW_SwitchCantileverFront_I5 AND NOT IX_HBW_SwitchCantileverBack_I6 THEN
                   QX_HBW_M4_CantileverBackward_Q8 := FALSE;
                   QX_HBW_M4_CantileverForward_Q7 := FALSE;
                   li_StepCase := 250;
               END_IF;

           250:
               gtyp_HBW.Vertical_Axis.di_Target_Position := ldi_PosRack_Vertical;
               gtyp_HBW.Vertical_Axis.x_Start_Positioning := TRUE;

               IF (gtyp_HBW.Vertical_Axis.di_Actual_Position <= (ldi_PosRack_Vertical + gtyp_HBW.Vertical_Axis.Config.di_Pos_Window))
                   AND (gtyp_HBW.Vertical_Axis.di_Actual_Position >= (ldi_PosRack_Vertical - gtyp_HBW.Vertical_Axis.Config.di_Pos_Window))
                   AND gtyp_HBW.Vertical_Axis.x_Position_Reached THEN
                   IF lx_Storage THEN
                       li_Return_LDT := RD_SYS_T(ldt_MQTT);
                       gtyp_HBW.History[3].i_code := 300;
                       gtyp_HBW.History[3].ldt_ts := DT_TO_LDT(ldt_MQTT);
                       gtyp_HBW.Rack_Workpiece[li_Counter_Act_Ver, li_Counter_Act_Hor] := gtyp_HBW.Workpiece;
                       gtyp_HBW.Rack_History[li_Counter_Act_Ver, li_Counter_Act_Hor].History := gtyp_HBW.History;
                       gtyp_Interface_Dashboard.Subscribe.State_HBW.x_active := FALSE;
                   ELSE
                       gtyp_HBW.Rack_Workpiece[li_Counter_Act_Ver, li_Counter_Act_Hor].s_id := '0';
                   END_IF;
                   gtyp_HBW.Vertical_Axis.x_Start_Positioning := FALSE;
                   li_StepCase := 260;
               END_IF;

           260:

               QX_HBW_M4_CantileverBackward_Q8 := TRUE;
               QX_HBW_M4_CantileverForward_Q7 := FALSE;

               IF NOT IX_HBW_SwitchCantileverFront_I5 AND IX_HBW_SwitchCantileverBack_I6 THEN
                   QX_HBW_M4_CantileverBackward_Q8 := FALSE;
                   QX_HBW_M4_CantileverForward_Q7 := FALSE;
                   li_StepCase := 0;
                   lx_Storage := FALSE;
               END_IF;

       ELSE
           ;
       END_CASE;


       IF gtyp_Setup.x_Clean_Rack_HBW THEN
           FOR li_Counter_Hor := 1 TO 3 DO
               FOR li_Counter_Ver := 1 TO 3 DO
                   gtyp_HBW.Rack_Workpiece[li_Counter_Ver, li_Counter_Hor].s_id := '0';
                   gtyp_HBW.Rack_Workpiece[li_Counter_Ver, li_Counter_Hor].s_state := '';
                   gtyp_HBW.Rack_Workpiece[li_Counter_Ver, li_Counter_Hor].s_type := '';
                   FOR li_Counter := 1 TO 8 DO
                       gtyp_HBW.Rack_History[li_Counter_Ver, li_Counter_Hor].History[li_Counter].i_code := 0;
                       gtyp_HBW.Rack_History[li_Counter_Ver, li_Counter_Hor].History[li_Counter].ldt_ts := DT#1990-01-01-00:00:00.00;
                   END_FOR;
               END_FOR;
           END_FOR;
           gtyp_Setup.x_Clean_Rack_HBW := FALSE;
       END_IF;


       QW_HBW_PWM_ConveyorBelt_M1   := gtyp_HBW.i_PWM_ConveyorBelt;
       QW_HBW_PWM_Cantilever_M4     := gtyp_HBW.i_PWM_Cantilever;
   ELSE
       FOR li_Counter_Hor := 1 TO 3 DO
           FOR li_Counter_Ver := 1 TO 3 DO
               IF gtyp_HBW.Rack_Workpiece[li_Counter_Ver, li_Counter_Hor].s_id = '' THEN
                   gtyp_HBW.Rack_Workpiece[li_Counter_Ver, li_Counter_Hor].s_id := '0';
                   gtyp_HBW.Rack_Workpiece[li_Counter_Ver, li_Counter_Hor].s_state := '';
                   gtyp_HBW.Rack_Workpiece[li_Counter_Ver, li_Counter_Hor].s_type := '';
                   FOR li_Counter := 1 TO 8 DO
                       gtyp_HBW.Rack_History[li_Counter_Ver, li_Counter_Hor].History[li_Counter].i_code := 0;
                       gtyp_HBW.Rack_History[li_Counter_Ver, li_Counter_Hor].History[li_Counter].ldt_ts := DT#1990-01-01-00:00:00.00;
                   END_FOR;
               END_IF;
           END_FOR;
       END_FOR;

       gtyp_HBW.x_Start_Park_Position := FALSE;
       gtyp_HBW.x_Park_Position_Reached := FALSE;
       gtyp_HBW.x_HBW_PickedUp_Accepted := FALSE;
       gtyp_HBW.x_HBW_Discards_Accepted := FALSE;
       gtyp_HBW.x_HBW_PickUp_Ready := FALSE;
       gtyp_HBW.x_HBW_Container_Available := FALSE;
       gtyp_HBW.x_Error := FALSE;

       li_Lights              := 1;
       lx_Start_TON_Fill_HBW  := TRUE;
       lx_Init                := TRUE;
   END_IF;
END_FUNCTION_BLOCK

FUNCTION_BLOCK PRG_VGR_Axis_rotate
   VAR
      lx_Init : Bool;
      lfb_rotate_Axis : FB_Axis;
   END_VAR



   IF lx_Init THEN


       lfb_rotate_Axis(ini_Axis           := 3,
                   indi_Increment          := gtyp_VGR.rotate_Axis.di_Increment,
                   inx_Ref_Switch          := IX_VGR_RefSwitchRotate_I3,
                   inx_Referencing         := gtyp_VGR.rotate_Axis.x_Reference,
                   inx_Start_Positioning   := gtyp_VGR.rotate_Axis.x_Start_Positioning,
                   indi_Target_Position    := gtyp_VGR.rotate_Axis.di_Target_Position,
                   ini_PWM                 := gtyp_VGR.rotate_Axis.i_PWM,
                   inouttyp_Config         := gtyp_VGR.rotate_Axis.Config,
                   inouttyp_Setup          := gtyp_SetupAxis);

       QX_VGR_M3_RotateClockwise_Q5          := lfb_rotate_Axis.outx_Motor_Neg;
       QX_VGR_M3_RotateCounterclockwise_Q6   := lfb_rotate_Axis.outx_Motor_Pos;
       QW_VGR_PWM_Rotate_M3                  := lfb_rotate_Axis.outi_Motor_PWM;
       gtyp_VGR.rotate_Axis.di_Actual_Position := lfb_rotate_Axis.outdi_Actual_Position;
       gtyp_VGR.rotate_Axis.x_Referenced       := lfb_rotate_Axis.outx_Referenced;
       gtyp_VGR.rotate_Axis.x_Position_Reached := lfb_rotate_Axis.outx_Position_Reached;
   ELSE
       lx_Init := TRUE;
   END_IF;
END_FUNCTION_BLOCK

FUNCTION_BLOCK PRG_SSC_Calibration_Color
   VAR
      lx_Init : Bool;
      lx_Start_TON_Wait : Bool;
      lx_Start_Positioning_m : Bool;
      lt_TON_Wait : Time;
      li_StepCase : Int;
      ldi_Pos_Horizontal : DInt;
      ldi_Pos_Vertical : DInt;
      lfb_R_Trig_Deaktivate : R_TRIG;
      lfb_TON_Wait : TON_TIME;
   END_VAR



   IF lx_Init THEN


       lfb_TON_Wait(IN := lx_Start_TON_Wait,
                     PT := lt_TON_Wait);

       lfb_R_Trig_Deaktivate(CLK:= NOT gtyp_Setup.x_Color_Sensor_Calibration
                              OR NOT (gtyp_Setup.i_Color_Sensor_Selection = 1));

       IF lfb_R_Trig_Deaktivate.Q THEN
           gtyp_Setup.x_Calculate_Value_Color := FALSE;
           gtyp_Setup.x_Set_Calib_Value_Color_Blue := FALSE;
           gtyp_Setup.x_Set_Calib_Value_Color_Red := FALSE;
           gtyp_Setup.x_Set_Calib_Value_Color_White := FALSE;
           gtyp_Setup.w_Calib_ColorValue_Blue := 0;
           gtyp_Setup.w_Calib_ColorValue_Red := 0;
           gtyp_Setup.w_Calib_ColorValue_White := 0;
           gtyp_Setup.w_Threshold_Red_Blue := 0;
           gtyp_Setup.w_Threshold_White_Red := 0;
           li_StepCase            := 0;
       END_IF;


       CASE li_StepCase OF

           0:
               lx_Start_TON_Wait := FALSE;
               li_StepCase := 10;

           10:
               IF gtyp_Setup.x_Color_Sensor_Calibration
                   AND (gtyp_Setup.i_Color_Sensor_Selection = 1) THEN
                   gtyp_Setup.x_Calculate_Value_Color := FALSE;
                   gtyp_Setup.x_Set_Calib_Value_Color_Blue := FALSE;
                   gtyp_Setup.x_Set_Calib_Value_Color_Red := FALSE;
                   gtyp_Setup.x_Set_Calib_Value_Color_White := FALSE;
                   gtyp_Setup.w_Calib_ColorValue_Blue := 0;
                   gtyp_Setup.w_Calib_ColorValue_Red := 0;
                   gtyp_Setup.w_Calib_ColorValue_White := 0;
                   gtyp_Setup.w_Threshold_Red_Blue := 0;
                   gtyp_Setup.w_Threshold_White_Red := 0;
                   li_StepCase := 20;
               END_IF;

           20:


               IF gtyp_Setup.x_Set_Calib_Value_Color_Blue THEN
                   gtyp_Setup.w_Calib_ColorValue_Blue := IW_SSC_ColorSensor_A1;
                   gtyp_Setup.x_Set_Calib_Value_Color_Blue := FALSE;
               ELSIF gtyp_Setup.x_Set_Calib_Value_Color_Red THEN
                   gtyp_Setup.w_Calib_ColorValue_Red := IW_SSC_ColorSensor_A1;
                   gtyp_Setup.x_Set_Calib_Value_Color_Red := FALSE;
               ELSIF gtyp_Setup.x_Set_Calib_Value_Color_White THEN
                   gtyp_Setup.w_Calib_ColorValue_White := IW_SSC_ColorSensor_A1;
                   gtyp_Setup.x_Set_Calib_Value_Color_White := FALSE;
               END_IF;

               gtyp_Setup.w_Threshold_White_Red  := gtyp_Setup.w_Calib_ColorValue_White + ((gtyp_Setup.w_Calib_ColorValue_Red - gtyp_Setup.w_Calib_ColorValue_White) / 2);
               gtyp_Setup.w_Threshold_Red_Blue   := gtyp_Setup.w_Calib_ColorValue_Red + ((gtyp_Setup.w_Calib_ColorValue_Blue - gtyp_Setup.w_Calib_ColorValue_Red) / 2);

               IF gtyp_Setup.x_Calculate_Value_Color THEN
                   gtyp_SSC.w_Threshold_White_Red := gtyp_Setup.w_Threshold_White_Red;
                   gtyp_SSC.w_Threshold_Red_Blue := gtyp_Setup.w_Threshold_Red_Blue;
                   gtyp_Setup.x_Calculate_Value_Color := FALSE;
               END_IF;


           ELSE
               ;
       END_CASE;

       IF (gtyp_Setup.i_Color_Sensor_Selection = 1) THEN

           gtyp_Setup.w_Actual_ColorValue := IW_SSC_ColorSensor_A1;
       END_IF;
   ELSE
       lx_Init := TRUE;
   END_IF;
END_FUNCTION_BLOCK

FUNCTION_BLOCK PRG_VGR_Axis_horizontal
   VAR
      lx_Init : Bool;
      lfb_horizontal_Axis : FB_Axis;
   END_VAR



   IF lx_Init THEN


       lfb_horizontal_Axis(ini_Axis       := 1,
                   indi_Increment          := gtyp_VGR.horizontal_Axis.di_Increment,
                   inx_Ref_Switch          := IX_VGR_RefSwitchHorizontalAxis_I2,
                   inx_Referencing         := gtyp_VGR.horizontal_Axis.x_Reference,
                   inx_Start_Positioning   := gtyp_VGR.horizontal_Axis.x_Start_Positioning,
                   indi_Target_Position    := gtyp_VGR.horizontal_Axis.di_Target_Position,
                   ini_PWM                 := gtyp_VGR.horizontal_Axis.i_PWM,
                   inouttyp_Config         := gtyp_VGR.horizontal_Axis.Config,
                   inouttyp_Setup          := gtyp_SetupAxis);

       QX_VGR_M2_HorizontalAxisForward_Q4    := lfb_horizontal_Axis.outx_Motor_Pos;
       QX_VGR_M2_HorizontalAxisBackward_Q3   := lfb_horizontal_Axis.outx_Motor_Neg;
       QW_VGR_PWM_Horizontal_M2              := lfb_horizontal_Axis.outi_Motor_PWM;
       gtyp_VGR.horizontal_Axis.di_Actual_Position    := lfb_horizontal_Axis.outdi_Actual_Position;
       gtyp_VGR.horizontal_Axis.x_Referenced          := lfb_horizontal_Axis.outx_Referenced;
       gtyp_VGR.horizontal_Axis.x_Position_Reached    := lfb_horizontal_Axis.outx_Position_Reached;
   ELSE
       lx_Init := TRUE;
   END_IF;
END_FUNCTION_BLOCK

FUNCTION_BLOCK PRG_MPO_Ablauf
   VAR
      lx_Init : Bool;
      lx_Start_TON_Wait : Bool;
      lx_Time_Error : Bool;
      lt_TON_Wait : Time;
      lx_Start_TON_State : Bool;
      ldt_MQTT : Date_And_Time;
      li_Return_LDT : Int;
      li_StepCase : Int;
      li_Lights : Int;
      li_Lights_old : Int;
      li_Counter : Int;
      lfb_blinker : FB_Blinker;
      lfb_TOF_ConveyerBelt_Out : TOF_TIME;
      lfb_TON_Wait : TON_TIME;
      lfb_TON_Error : TON_TIME;
      lfb_TON_State : TON_TIME;
      lfb_F_Trig_ConveyerBelt : F_TRIG;
   END_VAR



   IF lx_Init THEN


       lfb_TON_State(IN := NOT lx_Start_TON_State,
                       PT := T#2s);


       lfb_TON_Error(IN := lx_Time_Error,
                      PT := T#30s);


       IF (lfb_TON_State.Q OR (li_Lights <> li_Lights_old)) AND NOT lx_Start_TON_State THEN
           li_Lights_old := li_Lights;
           lx_Start_TON_State := TRUE;
           li_Return_LDT := RD_SYS_T(ldt_MQTT);
           gtyp_Interface_Dashboard.Subscribe.State_MPO.ldt_ts        := DT_TO_LDT(ldt_MQTT);
           gtyp_Interface_Dashboard.Subscribe.State_MPO.i_code        := li_Lights;
           gtyp_Interface_Dashboard.Subscribe.State_MPO.s_description := '';
           gtyp_Interface_Dashboard.Subscribe.State_MPO.s_station     := 'mpo';
           gtyp_Interface_Dashboard.Subscribe.State_MPO.s_target      := '';
       END_IF;


       IF NOT lfb_TON_State.Q AND lx_Start_TON_State THEN
           lx_Start_TON_State := FALSE;
       END_IF;


       lfb_TON_Wait(IN := lx_Start_TON_Wait,
                       PT := lt_TON_Wait);


      lfb_F_Trig_ConveyerBelt(CLK := NOT IX_MPO_LightBarrierEndOfConBelt_I3);


      lfb_TOF_ConveyerBelt_Out(IN:= lfb_F_Trig_ConveyerBelt.Q,
                                PT:= T#5000ms);


       lfb_blinker(int_periodendauer:= T#1000ms);


       CASE li_StepCase OF

           0:
               lx_Start_TON_Wait := FALSE;
               lx_Time_Error := FALSE;

               IF NOT gtyp_MPO.x_Error AND NOT gtyp_MPO.x_Start_Park_Position THEN
                   li_StepCase := 10;
               END_IF;

           10:
               li_Lights := 2;
               QX_MPO_LightOven_Q9   := FALSE;
               QX_MPO_Compressor_Q10 := TRUE;

               lx_Start_TON_Wait := TRUE;
               lt_TON_Wait := T#500ms;

               IF lfb_TON_Wait.Q THEN
                   lx_Start_TON_Wait := FALSE;
                   li_StepCase := 20;
               END_IF;

           20:
               QX_MPO_ValveOvenDoor_Q13 := TRUE;
               QX_MPO_ValveLowering_Q12 := FALSE;

               lx_Start_TON_Wait := TRUE;
               lt_TON_Wait := T#2000ms;

               IF lfb_TON_Wait.Q THEN
                   lx_Start_TON_Wait := FALSE;
                   li_StepCase := 30;
               END_IF;

           30:
               IF IX_MPO_RefSwitchOvenFeederOutside_I7 OR NOT IX_MPO_RefSwitchOvenFeederInside_I6 THEN
                   QX_MPO_M4_OvenFeederRetract_Q5 := TRUE;
                   QX_MPO_M4_OvenFeederExtend_Q6 := FALSE;
               ELSIF NOT IX_MPO_RefSwitchOvenFeederOutside_I7 AND IX_MPO_RefSwitchOvenFeederInside_I6 THEN
                   QX_MPO_M4_OvenFeederRetract_Q5 := FALSE;
                   QX_MPO_M4_OvenFeederExtend_Q6 := FALSE;
                   li_StepCase := 40;
               END_IF;

           40:

               QX_MPO_ValveOvenDoor_Q13 := FALSE;

               QX_MPO_M5_VacuumTowardsTurnTable_Q8 := TRUE;
               QX_MPO_M5_VacuumTowardsOven_Q7 := FALSE;
               QX_MPO_ValveVacuum_Q11        := FALSE;

               IF IX_MPO_RefSwitchVac_PosOven_I8 OR NOT IX_MPO_RefSwitchVac_PosTurnTable_I5 THEN
                   QX_MPO_M5_VacuumTowardsTurnTable_Q8 := TRUE;
                   QX_MPO_M5_VacuumTowardsOven_Q7 := FALSE;
               ELSIF NOT IX_MPO_RefSwitchVac_PosOven_I8 AND IX_MPO_RefSwitchVac_PosTurnTable_I5 THEN
                   QX_MPO_M5_VacuumTowardsTurnTable_Q8 := FALSE;
                   QX_MPO_M5_VacuumTowardsOven_Q7 := FALSE;
                   li_StepCase := 50;
               END_IF
               ;

           50:
               QX_MPO_M3_Saw_Q4 := FALSE;
               QX_MPO_ValveFeeder_Q14 := FALSE;
               QX_MPO_M2_ConveyorBeltForward_Q3 := FALSE;

               IF IX_MPO_RefSwitchTurnTable_PosSaw_I4 OR IX_MPO_RefSwitchTurnTable_PosBelt_I2 OR NOT IX_MPO_RefSwitchTurnTable_PosVac_I1 THEN
                   QX_MPO_M1_TurnTableClockwise_Q1 := FALSE;
                   QX_MPO_M1_TurnTableCounterclockwise_Q2 := TRUE;
               ELSIF NOT IX_MPO_RefSwitchTurnTable_PosSaw_I4 AND NOT IX_MPO_RefSwitchTurnTable_PosBelt_I2 AND IX_MPO_RefSwitchTurnTable_PosVac_I1 THEN
                   QX_MPO_M1_TurnTableClockwise_Q1 := FALSE;
                   QX_MPO_M1_TurnTableCounterclockwise_Q2 := FALSE;
                   QX_MPO_Compressor_Q10 := FALSE;
                   li_StepCase := 60;
               END_IF;

           60:
               li_Lights := 1;
               IF gtyp_VGR.x_MPO_Req_Discard THEN
                   li_Lights := 2;
                   QX_MPO_Compressor_Q10 := TRUE;
                   li_StepCase := 70;
               END_IF;

           70:
               lx_Start_TON_Wait := TRUE;
               lt_TON_Wait := T#500ms;

               IF lfb_TON_Wait.Q THEN
                   lx_Start_TON_Wait := FALSE;
                   li_StepCase := 80;
               END_IF;

           80:
               QX_MPO_ValveOvenDoor_Q13 := TRUE;

               lx_Start_TON_Wait := TRUE;
               lt_TON_Wait := T#2000ms;

               IF lfb_TON_Wait.Q THEN
                   lx_Start_TON_Wait := FALSE;
                   li_StepCase := 90;
               END_IF;

           90:
               QX_MPO_M4_OvenFeederRetract_Q5    := FALSE;
               QX_MPO_M4_OvenFeederExtend_Q6     := TRUE;

               IF IX_MPO_RefSwitchOvenFeederOutside_I7 AND NOT IX_MPO_RefSwitchOvenFeederInside_I6 THEN
                   QX_MPO_M4_OvenFeederRetract_Q5 := FALSE;
                   QX_MPO_M4_OvenFeederExtend_Q6 := FALSE;
                   gtyp_MPO.x_MPO_Discards_Accepted := FALSE;
                   gtyp_MPO.x_Discard_Ready      := TRUE;
                   li_StepCase := 100;
               END_IF;

           100:

               lx_Time_Error := TRUE;

               IF gtyp_VGR.x_MPO_Discards AND NOT IX_MPO_LightBarrierOven_I9 THEN
                   gtyp_Interface_Dashboard.Subscribe.State_MPO.x_active := TRUE;
                   gtyp_MPO.History  := gtyp_VGR.History;
                   gtyp_MPO.Workpiece := gtyp_VGR.Workpiece;
                   gtyp_MPO.x_Discard_Ready := FALSE;
                   gtyp_MPO.x_MPO_Discards_Accepted := TRUE;
                   lx_Time_Error := FALSE;
                   li_StepCase := 105;
               END_IF;


               IF lfb_TON_Error.Q THEN
                   li_Lights := 4;
                   lx_Time_Error := FALSE;
                   gtyp_Interface_Dashboard.Subscribe.State_Order.ldt_ts := DT_TO_LDT(ldt_MQTT);
                   gtyp_Interface_Dashboard.Subscribe.State_Order.s_state := 'WAITING_FOR_ORDER';
                   gtyp_Interface_Dashboard.Subscribe.State_Order.s_type := '';
                   gtyp_Interface_Dashboard.Subscribe.State_MPO.x_active := FALSE;
                   gtyp_MPO.x_Discard_Ready := FALSE;
                   gtyp_MPO.x_MPO_Discards_Accepted := FALSE;
                   gtyp_MPO.x_Error := TRUE;
                   li_StepCase := 0;
               END_IF;

           105:
               IF NOT gtyp_VGR.x_MPO_Discards AND IX_MPO_RefSwitchOvenFeederOutside_I7 AND NOT IX_MPO_RefSwitchOvenFeederInside_I6 THEN
                   gtyp_MPO.x_MPO_Discards_Accepted := FALSE;
                   QX_MPO_M4_OvenFeederRetract_Q5 := TRUE;
                   QX_MPO_M4_OvenFeederExtend_Q6 := FALSE;
                   li_StepCase := 110;
               END_IF;

           110:
               IF NOT IX_MPO_RefSwitchOvenFeederOutside_I7 AND IX_MPO_RefSwitchOvenFeederInside_I6 THEN
                   QX_MPO_M4_OvenFeederRetract_Q5 := FALSE;
                   QX_MPO_M4_OvenFeederExtend_Q6 := FALSE;
                   li_StepCase := 120;
               END_IF;

           120:
               QX_MPO_ValveOvenDoor_Q13 := FALSE;

               lx_Start_TON_Wait := TRUE;
               lt_TON_Wait := T#2000ms;

               IF lfb_TON_Wait.Q THEN
                   lx_Start_TON_Wait := FALSE;
                   li_StepCase := 130;
               END_IF;

           130:
               QX_MPO_LightOven_Q9:= lfb_blinker.outx_blinker;

               IF NOT gtyp_VGR.x_MPO_Discards THEN
                   li_Return_LDT := RD_SYS_T(ldt_MQTT);
                   gtyp_MPO.History[5].i_code := 500;
                   gtyp_MPO.History[5].ldt_ts := DT_TO_LDT(ldt_MQTT);

                   QX_MPO_M5_VacuumTowardsOven_Q7 := TRUE;
                   QX_MPO_M5_VacuumTowardsTurnTable_Q8 := FALSE;

                   IF NOT IX_MPO_RefSwitchVac_PosTurnTable_I5 AND IX_MPO_RefSwitchVac_PosOven_I8 THEN
                       QX_MPO_M5_VacuumTowardsOven_Q7 := FALSE;
                       QX_MPO_M5_VacuumTowardsTurnTable_Q8 := FALSE;
                   END_IF;
               END_IF;

               lx_Start_TON_Wait := TRUE;
               lt_TON_Wait := T#4000ms;

               IF lfb_TON_Wait.Q THEN
                   lx_Start_TON_Wait := FALSE;
                   li_StepCase := 140;
               END_IF;

           140:
               QX_MPO_LightOven_Q9       := FALSE;
               QX_MPO_ValveOvenDoor_Q13  := TRUE;

               IF NOT gtyp_VGR.x_MPO_Discards THEN
                   QX_MPO_M5_VacuumTowardsOven_Q7 := TRUE;
                   QX_MPO_M5_VacuumTowardsTurnTable_Q8 := FALSE;

                   IF NOT IX_MPO_RefSwitchVac_PosTurnTable_I5 AND IX_MPO_RefSwitchVac_PosOven_I8 THEN
                       QX_MPO_M5_VacuumTowardsOven_Q7 := FALSE;
                       QX_MPO_M5_VacuumTowardsTurnTable_Q8 := FALSE;
                   END_IF;
               END_IF;

               lx_Start_TON_Wait := TRUE;
               lt_TON_Wait := T#2000ms;

               IF lfb_TON_Wait.Q THEN
                   lx_Start_TON_Wait := FALSE;
                   li_StepCase := 150;
               END_IF;

           150:

               QX_MPO_M4_OvenFeederRetract_Q5 := FALSE;
               QX_MPO_M4_OvenFeederExtend_Q6 := TRUE;

               IF NOT gtyp_VGR.x_MPO_Discards THEN
                   QX_MPO_M5_VacuumTowardsOven_Q7 := TRUE;
                   QX_MPO_M5_VacuumTowardsTurnTable_Q8 := FALSE;

                   IF NOT IX_MPO_RefSwitchVac_PosTurnTable_I5 AND IX_MPO_RefSwitchVac_PosOven_I8 THEN
                       QX_MPO_M5_VacuumTowardsOven_Q7 := FALSE;
                       QX_MPO_M5_VacuumTowardsTurnTable_Q8 := FALSE;
                   END_IF;
               END_IF;

               IF IX_MPO_RefSwitchOvenFeederOutside_I7 AND NOT IX_MPO_RefSwitchOvenFeederInside_I6 THEN
                   QX_MPO_M4_OvenFeederRetract_Q5 := FALSE;
                   QX_MPO_M4_OvenFeederExtend_Q6 := FALSE;
               END_IF;

               IF IX_MPO_RefSwitchOvenFeederOutside_I7 AND NOT IX_MPO_RefSwitchOvenFeederInside_I6
                   AND NOT IX_MPO_RefSwitchVac_PosTurnTable_I5 AND IX_MPO_RefSwitchVac_PosOven_I8 THEN
                   QX_MPO_M5_VacuumTowardsOven_Q7 := FALSE;
                   QX_MPO_M5_VacuumTowardsTurnTable_Q8 := FALSE;
                   QX_MPO_M4_OvenFeederRetract_Q5 := FALSE;
                   QX_MPO_M4_OvenFeederExtend_Q6 := FALSE;
                   li_StepCase := 160;
               END_IF;

           160:
               QX_MPO_ValveLowering_Q12:= TRUE;

               lx_Start_TON_Wait := TRUE;
               lt_TON_Wait := T#1000ms;

               IF lfb_TON_Wait.Q THEN
                   lx_Start_TON_Wait := FALSE;
                   li_StepCase := 170;
               END_IF;

           170:
               QX_MPO_ValveVacuum_Q11:= TRUE;

               lx_Start_TON_Wait := TRUE;
               lt_TON_Wait := T#1000ms;

               IF lfb_TON_Wait.Q THEN
                   lx_Start_TON_Wait := FALSE;
                   li_StepCase := 180;
               END_IF;

           180:
               QX_MPO_ValveLowering_Q12 := FALSE;

               lx_Start_TON_Wait := TRUE;
               lt_TON_Wait := T#1000ms;

               IF lfb_TON_Wait.Q THEN
                   lx_Start_TON_Wait := FALSE;
                   li_StepCase := 190;
               END_IF;

           190:
               QX_MPO_M4_OvenFeederRetract_Q5 := TRUE;
               QX_MPO_M4_OvenFeederExtend_Q6 := FALSE;
               QX_MPO_M5_VacuumTowardsOven_Q7 := FALSE;
               QX_MPO_M5_VacuumTowardsTurnTable_Q8 := TRUE;

               IF IX_MPO_RefSwitchVac_PosTurnTable_I5 AND NOT IX_MPO_RefSwitchVac_PosOven_I8 THEN
                   QX_MPO_M5_VacuumTowardsOven_Q7 := FALSE;
                   QX_MPO_M5_VacuumTowardsTurnTable_Q8 := FALSE;
               END_IF;

               IF NOT IX_MPO_RefSwitchOvenFeederOutside_I7 AND IX_MPO_RefSwitchOvenFeederInside_I6 THEN
                   QX_MPO_M4_OvenFeederRetract_Q5 := FALSE;
                   QX_MPO_M4_OvenFeederExtend_Q6 := FALSE;
               END_IF;

               IF NOT IX_MPO_RefSwitchOvenFeederOutside_I7 AND IX_MPO_RefSwitchOvenFeederInside_I6
                   AND IX_MPO_RefSwitchVac_PosTurnTable_I5 AND NOT IX_MPO_RefSwitchVac_PosOven_I8 THEN
                   QX_MPO_M5_VacuumTowardsOven_Q7 := FALSE;
                   QX_MPO_M5_VacuumTowardsTurnTable_Q8 := FALSE;
                   QX_MPO_M4_OvenFeederRetract_Q5 := FALSE;
                   QX_MPO_M4_OvenFeederExtend_Q6 := FALSE;
                   QX_MPO_ValveOvenDoor_Q13 := FALSE;
                   li_StepCase := 200;
               END_IF;

           200:
               IF IX_MPO_RefSwitchTurnTable_PosVac_I1 THEN
                   QX_MPO_ValveLowering_Q12 := TRUE;

                   lx_Start_TON_Wait := TRUE;
                   lt_TON_Wait := T#2000ms;

                   IF lfb_TON_Wait.Q THEN
                       lx_Start_TON_Wait := FALSE;
                       li_StepCase := 210;
                   END_IF;
               END_IF;

           210:
               QX_MPO_ValveVacuum_Q11 := FALSE;

               lx_Start_TON_Wait := TRUE;
               lt_TON_Wait := T#2000ms;

               IF lfb_TON_Wait.Q THEN
                   lx_Start_TON_Wait := FALSE;
                   li_StepCase := 220;
               END_IF;

           220:
               QX_MPO_ValveLowering_Q12 := FALSE;

               lx_Start_TON_Wait := TRUE;
               lt_TON_Wait := T#2000ms;

               IF lfb_TON_Wait.Q THEN
                   lx_Start_TON_Wait := FALSE;
                   li_StepCase := 230;
               END_IF;

           230:
               IF NOT IX_MPO_RefSwitchTurnTable_PosSaw_I4 AND NOT IX_MPO_RefSwitchTurnTable_PosBelt_I2 AND IX_MPO_RefSwitchTurnTable_PosVac_I1 THEN
                   QX_MPO_M1_TurnTableClockwise_Q1 := TRUE;
                   QX_MPO_M1_TurnTableCounterclockwise_Q2 := FALSE;
               ELSIF IX_MPO_RefSwitchTurnTable_PosSaw_I4 OR IX_MPO_RefSwitchTurnTable_PosBelt_I2 AND NOT IX_MPO_RefSwitchTurnTable_PosVac_I1 THEN
                   QX_MPO_M1_TurnTableClockwise_Q1 := FALSE;
                   QX_MPO_M1_TurnTableCounterclockwise_Q2 := FALSE;
                   li_StepCase := 240;
               END_IF;

           240:
               QX_MPO_M3_Saw_Q4 := TRUE;

               lx_Start_TON_Wait := TRUE;
               lt_TON_Wait := T#4000ms;

               IF lfb_TON_Wait.Q THEN
                   li_Return_LDT := RD_SYS_T(ldt_MQTT);
                   gtyp_MPO.History[6].i_code := 600;
                   gtyp_MPO.History[6].ldt_ts := DT_TO_LDT(ldt_MQTT);

                   lx_Start_TON_Wait := FALSE;
                   QX_MPO_M3_Saw_Q4 := FALSE;
                   li_StepCase := 250;
               END_IF;

           250:
               IF IX_MPO_RefSwitchTurnTable_PosSaw_I4 AND NOT IX_MPO_RefSwitchTurnTable_PosBelt_I2 AND NOT IX_MPO_RefSwitchTurnTable_PosVac_I1 THEN
                   QX_MPO_M1_TurnTableClockwise_Q1 := TRUE;
                   QX_MPO_M1_TurnTableCounterclockwise_Q2 := FALSE;
               ELSIF NOT IX_MPO_RefSwitchTurnTable_PosSaw_I4 AND IX_MPO_RefSwitchTurnTable_PosBelt_I2 AND NOT IX_MPO_RefSwitchTurnTable_PosVac_I1 THEN
                   QX_MPO_M1_TurnTableClockwise_Q1 := FALSE;
                   QX_MPO_M1_TurnTableCounterclockwise_Q2 := FALSE;
                   li_StepCase := 260;
               END_IF;

           260:
               QX_MPO_ValveFeeder_Q14 := TRUE;

               lx_Start_TON_Wait := TRUE;
               lt_TON_Wait := T#1000ms;

               IF lfb_TON_Wait.Q THEN
                   lx_Start_TON_Wait := FALSE;
                   QX_MPO_ValveFeeder_Q14 := FALSE;
                   QX_MPO_Compressor_Q10 := FALSE;
                   li_StepCase := 270;
               END_IF;

           270:
               IF IX_MPO_RefSwitchTurnTable_PosSaw_I4 OR IX_MPO_RefSwitchTurnTable_PosBelt_I2 OR NOT IX_MPO_RefSwitchTurnTable_PosVac_I1 THEN
                   QX_MPO_M1_TurnTableClockwise_Q1 := FALSE;
                   QX_MPO_M1_TurnTableCounterclockwise_Q2 := TRUE;
               ELSIF NOT IX_MPO_RefSwitchTurnTable_PosSaw_I4 AND NOT IX_MPO_RefSwitchTurnTable_PosBelt_I2 AND IX_MPO_RefSwitchTurnTable_PosVac_I1 THEN
                   QX_MPO_M1_TurnTableClockwise_Q1 := FALSE;
                   QX_MPO_M1_TurnTableCounterclockwise_Q2 := FALSE;
                   QX_MPO_Compressor_Q10 := FALSE;
                   li_StepCase := 280;
               END_IF;

           280:
               QX_MPO_M2_ConveyorBeltForward_Q3 := TRUE;

               lx_Time_Error := TRUE;

               IF lfb_TOF_ConveyerBelt_Out.Q THEN
                   gtyp_SLD.History  := gtyp_MPO.History;
                   gtyp_SLD.Workpiece := gtyp_MPO.Workpiece;
                   gtyp_MPO.Workpiece.s_id := '0';
                   gtyp_MPO.Workpiece.s_state := '';
                   gtyp_MPO.Workpiece.s_type := '';
                   FOR li_Counter := 1 TO 8 DO
                       gtyp_MPO.History[li_Counter].i_code := 0;
                       gtyp_MPO.History[li_Counter].ldt_ts := DT#1990-01-01-00:00:00.00;
                   END_FOR;

                   gtyp_Interface_Dashboard.Subscribe.State_MPO.x_active := FALSE;

                   lx_Time_Error := FALSE;
                   li_StepCase := 290;
               END_IF;


               IF lfb_TON_Error.Q THEN
                   li_Lights := 4;
                   lx_Time_Error := FALSE;
                   QX_MPO_M2_ConveyorBeltForward_Q3 := FALSE;
                   gtyp_Interface_Dashboard.Subscribe.State_MPO.x_active := FALSE;
                   gtyp_MPO.x_Error := TRUE;
                   li_StepCase := 0;
               END_IF;

           290:

               IF NOT lfb_TOF_ConveyerBelt_Out.Q THEN
                   lx_Start_TON_Wait := FALSE;
                   QX_MPO_M2_ConveyorBeltForward_Q3 := FALSE;
                   li_StepCase := 60;
               END_IF;

           ELSE
               ;
       END_CASE;

       QW_MPO_PWM_TurnTable_M1   := gtyp_MPO.i_PWM_TurnTable;
       QW_MPO_PWM_Vacuum_M5      := gtyp_MPO.i_PWM_Vacuum;

   ELSE
       li_Lights := 1;
       lx_Init := TRUE;
       gtyp_MPO.x_Start_Park_Position := FALSE;
       gtyp_MPO.x_Park_Position_Reached := FALSE;
   END_IF;
END_FUNCTION_BLOCK

FUNCTION_BLOCK PRG_VGR_Axis_vertical
   VAR
      lx_Init : Bool;
      lfb_vertical_Axis : FB_Axis;
   END_VAR



   IF lx_Init THEN


       lfb_vertical_Axis(ini_Axis         := 2,
                   indi_Increment          := gtyp_VGR.vertical_Axis.di_Increment,
                   inx_Ref_Switch          := IX_VGR_RefSwitchVerticalAxis_I1,
                   inx_Referencing         := gtyp_VGR.vertical_Axis.x_Reference,
                   inx_Start_Positioning   := gtyp_VGR.vertical_Axis.x_Start_Positioning,
                   indi_Target_Position    := gtyp_VGR.vertical_Axis.di_Target_Position,
                   ini_PWM                 := gtyp_VGR.vertical_Axis.i_PWM,
                   inouttyp_Config         := gtyp_VGR.vertical_Axis.Config,
                   inouttyp_Setup          := gtyp_SetupAxis);

       QX_VGR_M1_VerticalAxisUp_Q1       := lfb_vertical_Axis.outx_Motor_Neg;
       QX_VGR_M1_VerticalAxisDown_Q2     := lfb_vertical_Axis.outx_Motor_Pos;
       QW_VGR_PWM_Vertical_M1            := lfb_vertical_Axis.outi_Motor_PWM;
       gtyp_VGR.vertical_Axis.di_Actual_Position:= lfb_vertical_Axis.outdi_Actual_Position;
       gtyp_VGR.vertical_Axis.x_Referenced      := lfb_vertical_Axis.outx_Referenced;
       gtyp_VGR.vertical_Axis.x_Position_Reached:= lfb_vertical_Axis.outx_Position_Reached;
   ELSE
       lx_Init := TRUE;
   END_IF;
END_FUNCTION_BLOCK

FUNCTION_BLOCK PRG_HBW_Axis_Vertical
   VAR
      lx_Init : Bool;
      lfb_Vertical_Axis : FB_Axis;
   END_VAR



   IF lx_Init THEN


       lfb_Vertical_Axis( ini_Axis                := 7,
                           indi_Increment          := gtyp_HBW.Vertical_Axis.di_Increment,
                           inx_Ref_Switch          := IX_HBW_RefSwitchVerticalAxis_I4,
                           inx_Referencing         := gtyp_HBW.Vertical_Axis.x_Reference,
                           inx_Start_Positioning   := gtyp_HBW.Vertical_Axis.x_Start_Positioning,
                           indi_Target_Position    := gtyp_HBW.Vertical_Axis.di_Target_Position,
                           ini_PWM                 := gtyp_HBW.Vertical_Axis.i_PWM,
                           inouttyp_Config         := gtyp_HBW.Vertical_Axis.Config,
                           inouttyp_Setup          := gtyp_SetupAxis);

       QX_HBW_M3_VerticalAxisDownward_Q5           := lfb_Vertical_Axis.outx_Motor_Pos;
       QX_HBW_M3_VerticalAxisUpward_Q6             := lfb_Vertical_Axis.outx_Motor_Neg;
       QW_HBW_PWM_VerticalAxis_M3                  := lfb_Vertical_Axis.outi_Motor_PWM;
       gtyp_HBW.Vertical_Axis.di_Actual_Position   := lfb_Vertical_Axis.outdi_Actual_Position;
       gtyp_HBW.Vertical_Axis.x_Referenced         := lfb_Vertical_Axis.outx_Referenced;
       gtyp_HBW.Vertical_Axis.x_Position_Reached   := lfb_Vertical_Axis.outx_Position_Reached;
   ELSE
       lx_Init := TRUE;
   END_IF;
END_FUNCTION_BLOCK

FUNCTION_BLOCK PRG_DSI_Status
   VAR
      lx_Init : Bool;
      lx_Start : Bool;
      li_StepCase : Int;
      ldt_MQTT : Date_And_Time;
      li_Return_LDT : Int;
      lfb_R_Trig_Storage : R_TRIG;
      lfb_F_Trig_Storage : F_TRIG;
      lfb_TON_Status : TON_TIME;
      lx_StartStatus : Bool;
      lfb_TON_Schritt : TON_TIME;
      lx_StartTimer : Bool;
   END_VAR



   IF lx_Init THEN


       lfb_TON_Status(IN := NOT lx_StartStatus,
                       PT := T#2s);


       lfb_R_Trig_Storage(CLK := NOT IX_SSC_LightBarrierStorage_I3);
       lfb_F_Trig_Storage(CLK := NOT IX_SSC_LightBarrierStorage_I3);


       IF (lfb_TON_Status.Q OR lfb_R_Trig_Storage.Q OR lfb_F_Trig_Storage.Q) AND NOT lx_StartStatus THEN
           lx_StartStatus := TRUE;
           li_Return_LDT := RD_SYS_T(ldt_MQTT);
           IF NOT IX_SSC_LightBarrierStorage_I3 THEN
               gtyp_Interface_Dashboard.Subscribe.State_DSI.i_code := 0;
               gtyp_Interface_Dashboard.Subscribe.State_DSI.x_active := TRUE;
           ELSE
               gtyp_Interface_Dashboard.Subscribe.State_DSI.i_code := 1;
               IF lfb_F_Trig_Storage.Q THEN
                   gtyp_Interface_Dashboard.Subscribe.State_DSI.x_active := FALSE;
               END_IF;
           END_IF;
           gtyp_Interface_Dashboard.Subscribe.State_DSI.ldt_ts := DT_TO_LDT(ldt_MQTT);
           gtyp_Interface_Dashboard.Subscribe.State_DSI.s_station := 'dsi';
           gtyp_Interface_Dashboard.Subscribe.State_DSI.s_target := '';
           gtyp_Interface_Dashboard.Subscribe.State_DSI.s_description := '';
       END_IF;

       IF NOT lfb_TON_Status.Q AND lx_StartStatus THEN
           lx_StartStatus := FALSE;
       END_IF;
   ELSE
       lx_Init := TRUE;
   END_IF;
END_FUNCTION_BLOCK

FUNCTION_BLOCK PRG_SLD_Ablauf
   VAR
      lx_Init : Bool;
      lx_Start_TON_Wait : Bool;
      lx_Time_Error : Bool;
      lt_TON_Wait : Time;
      lx_Start_TON_State : Bool;
      ldt_MQTT : Date_And_Time;
      li_Return_LDT : Int;
      li_Lights : Int;
      li_Lights_old : Int;
      lw_ColorValueMin : Word;
      li_CounterActual : Int;
      lx_White : Bool;
      lx_Blue : Bool;
      lx_Red : Bool;
      li_StepCase : Int;
      ls_Color : String;
      lfb_TOF_ConveyerBelt_Out : TOF_TIME;
      lfb_TON_Wait : TON_TIME;
      lfb_TON_Error : TON_TIME;
      lfb_TON_State : TON_TIME;
      lfb_F_Trig_Counter : F_TRIG;
      lfb_R_Trig_Counter : R_TRIG;
   END_VAR



   IF lx_Init THEN


       IF gtyp_Setup.x_Color_Sensor_Calibration THEN
           li_StepCase := 0;
       END_IF;


       lfb_TON_State(IN := NOT lx_Start_TON_State,
                       PT := T#2s);


       IF (lfb_TON_State.Q OR (li_Lights <> li_Lights_old)) AND NOT lx_Start_TON_State THEN
           li_Lights_old := li_Lights;
           lx_Start_TON_State := TRUE;
           li_Return_LDT := RD_SYS_T(ldt_MQTT);
           gtyp_Interface_Dashboard.Subscribe.State_SLD.ldt_ts := DT_TO_LDT(ldt_MQTT);
           gtyp_Interface_Dashboard.Subscribe.State_SLD.i_code := li_Lights;
           gtyp_Interface_Dashboard.Subscribe.State_SLD.s_description := '';
           gtyp_Interface_Dashboard.Subscribe.State_SLD.s_station := 'sld';
           gtyp_Interface_Dashboard.Subscribe.State_SLD.s_target := '';
       END_IF;


       IF NOT lfb_TON_State.Q AND lx_Start_TON_State THEN
           lx_Start_TON_State := FALSE;
       END_IF;


       lfb_TON_Wait(IN := lx_Start_TON_Wait,
                        PT := lt_TON_Wait);


       lfb_TON_Error(IN:= lx_Time_Error,
                      PT:= T#30s);


       lfb_R_Trig_Counter(CLK:= IX_SLD_PulseCounter_I1);


       lfb_F_Trig_Counter(CLK := IX_SLD_PulseCounter_I1);


       CASE li_StepCase OF

           0:
               lx_Start_TON_Wait := FALSE;
               lx_Time_Error := FALSE;
               li_Lights := 1;

               IF NOT gtyp_SLD.x_Error AND NOT gtyp_Setup.x_Color_Sensor_Calibration THEN
                   li_StepCase := 10;
               END_IF;

           10:
               li_Lights := 2;
               QX_SLD_Compressor_Q2 := TRUE;

               lx_Start_TON_Wait := TRUE;
               lt_TON_Wait := T#1000ms;

               IF lfb_TON_Wait.Q THEN
                   lx_Start_TON_Wait := FALSE;
                   li_StepCase := 20;
               END_IF;

           20:
               QX_SLD_ValveFirstEjectorWhite_Q3  := FALSE;
               QX_SLD_ValveSecondEjectorRed_Q4   := FALSE;
               QX_SLD_ValveThirdEjectorBlue_Q5   := FALSE;
               QX_SLD_M1_ConveyorBelt_Q1         := FALSE;

               lx_Start_TON_Wait := TRUE;
               lt_TON_Wait := T#2000ms;

               IF lfb_TON_Wait.Q THEN
                   lx_Start_TON_Wait := FALSE;
                   li_StepCase := 30;
               END_IF;

           30:

               QX_SLD_Compressor_Q2 := FALSE;

               li_StepCase := 40;

           40:

               li_Lights := 1;
               IF NOT IX_SLD_LightBarrierInlet_I2 THEN
                   gtyp_Interface_Dashboard.Subscribe.State_SLD.x_active := TRUE;
                   li_Lights := 2;
                   QX_SLD_Compressor_Q2      := TRUE;
                   QX_SLD_M1_ConveyorBelt_Q1 := TRUE;
                   lw_ColorValueMin           := 40000;
                   li_CounterActual := 0;
                   lx_Blue := FALSE;
                   lx_Red := FALSE;
                   lx_White := FALSE;
                   li_StepCase := 50;
               END_IF;

           50:
               IF lw_ColorValueMin > IW_SLD_ColorSensor_A4 THEN
                   lw_ColorValueMin := IW_SLD_ColorSensor_A4;
               END_IF;

               lx_Time_Error := TRUE;


               IF NOT IX_SLD_LightBarrierBehindColorSensor_I3 THEN
                   lx_Time_Error  := FALSE;
                   li_StepCase    := 60;
               END_IF;


               IF lfb_TON_Error.Q THEN
                   li_Lights                  := 4;
                   lx_Time_Error              := FALSE;
                   QX_SLD_Compressor_Q2      := FALSE;
                   QX_SLD_M1_ConveyorBelt_Q1 := FALSE;
                   gtyp_Interface_Dashboard.Subscribe.State_SLD.x_active := FALSE;
                   gtyp_SLD.x_Error          := TRUE;
                   li_StepCase                := 0;
               END_IF;

           60:

               IF lw_ColorValueMin >= gtyp_SLD.w_Threshold_Red_Blue THEN
                   lx_Blue := TRUE;
               ELSIF lw_ColorValueMin <= gtyp_SLD.w_Threshold_White_Red THEN
                   lx_White := TRUE;
               ELSIF lw_ColorValueMin > gtyp_SLD.w_Threshold_White_Red AND lw_ColorValueMin < gtyp_SLD.w_Threshold_Red_Blue THEN
                   lx_Red := TRUE;
               END_IF;


               IF lfb_R_Trig_Counter.Q OR lfb_F_Trig_Counter.Q THEN
                   li_CounterActual := li_CounterActual + 1;
               END_IF;


               IF (li_CounterActual = gtyp_SLD.i_CounterValue_Blue) AND lx_Blue THEN
                   QX_SLD_ValveThirdEjectorBlue_Q5 := TRUE;
                   li_Return_LDT := RD_SYS_T(ldt_MQTT);
                   gtyp_SLD.Workpiece.s_state := 'PROCESSED';
                   gtyp_SLD.History[7].i_code := 700;
                   gtyp_SLD.History[7].ldt_ts := DT_TO_LDT(ldt_MQTT);
                   li_StepCase := 70;
               ELSIF (li_CounterActual = gtyp_SLD.i_CounterValue_White) AND lx_White THEN
                   QX_SLD_ValveFirstEjectorWhite_Q3 := TRUE;
                   li_Return_LDT := RD_SYS_T(ldt_MQTT);
                   gtyp_SLD.Workpiece.s_state := 'PROCESSED';
                   gtyp_SLD.History[7].i_code := 700;
                   gtyp_SLD.History[7].ldt_ts := DT_TO_LDT(ldt_MQTT);
                   li_StepCase := 70;
               ELSIF (li_CounterActual = gtyp_SLD.i_CounterValue_Red) AND lx_Red THEN
                   QX_SLD_ValveSecondEjectorRed_Q4 := TRUE;
                   li_Return_LDT := RD_SYS_T(ldt_MQTT);
                   gtyp_SLD.Workpiece.s_state := 'PROCESSED';
                   gtyp_SLD.History[7].i_code := 700;
                   gtyp_SLD.History[7].ldt_ts := DT_TO_LDT(ldt_MQTT);
                   li_StepCase := 70;
               ELSIF (li_CounterActual = 80) THEN
                   li_Lights := 4;
                   gtyp_SLD.x_Error := TRUE;
                   li_StepCase := 70;
               END_IF;

           70:
               lx_Start_TON_Wait := TRUE;
               lt_TON_Wait := T#500ms;

               IF lfb_TON_Wait.Q THEN
                   QX_SLD_ValveThirdEjectorBlue_Q5 := FALSE;
                   QX_SLD_ValveFirstEjectorWhite_Q3 := FALSE;
                   QX_SLD_ValveSecondEjectorRed_Q4 := FALSE;
                   lx_Start_TON_Wait := FALSE;
                   li_StepCase := 80;
               END_IF;

           80:

               lx_Start_TON_Wait := TRUE;
               lt_TON_Wait := T#2000ms;

               IF lfb_TON_Wait.Q THEN
                   QX_SLD_Compressor_Q2 := FALSE;
                   lx_Start_TON_Wait := FALSE;
                   li_StepCase := 90;
               END_IF;

           90:
               QX_SLD_M1_ConveyorBelt_Q1    := FALSE;
               li_StepCase := 40;

           ELSE
               ;
       END_CASE;

   ELSE
       gtyp_SLD.x_Error := FALSE;
       li_Lights := 1;
       lx_Init := TRUE;
   END_IF;
END_FUNCTION_BLOCK

FUNCTION_BLOCK PRG_HBW_Axis_Horizontal
   VAR
      lx_Init : Bool;
      lfb_Horizontal_Axis : FB_Axis;
   END_VAR



   IF lx_Init THEN


       lfb_Horizontal_Axis(ini_Axis               := 6,
                            indi_Increment          := gtyp_HBW.Horizontal_Axis.di_Increment,
                            inx_Ref_Switch         := IX_HBW_RefSwitchHorizontalAxis_I1,
                            inx_Referencing        := gtyp_HBW.Horizontal_Axis.x_Reference,
                            inx_Start_Positioning  := gtyp_HBW.Horizontal_Axis.x_Start_Positioning,
                            indi_Target_Position   := gtyp_HBW.Horizontal_Axis.di_Target_Position,
                            ini_PWM                := gtyp_HBW.Horizontal_Axis.i_PWM,
                            inouttyp_Config        := gtyp_HBW.Horizontal_Axis.Config,
                            inouttyp_Setup         := gtyp_SetupAxis);

       QX_HBW_M2_HorizontalTowardsRack_Q3            := lfb_Horizontal_Axis.outx_Motor_Pos;
       QX_HBW_M2_HorizontalTowardsConveyorBelt_Q4    := lfb_Horizontal_Axis.outx_Motor_Neg;
       QW_HBW_PWM_HorizontalAxis_M2                  := lfb_Horizontal_Axis.outi_Motor_PWM;
       gtyp_HBW.Horizontal_Axis.di_Actual_Position   := lfb_Horizontal_Axis.outdi_Actual_Position;
       gtyp_HBW.Horizontal_Axis.x_Referenced         := lfb_Horizontal_Axis.outx_Referenced;
       gtyp_HBW.Horizontal_Axis.x_Position_Reached   := lfb_Horizontal_Axis.outx_Position_Reached;
   ELSE
       lx_Init := TRUE;
   END_IF;
END_FUNCTION_BLOCK

FUNCTION_BLOCK PRG_SSC_Light
   VAR
      lx_Init : Bool;
      lx_Start : Bool;
      li_StepCase : Int;
      ldt_MQTT : Date_And_Time;
      lldt_ts_old : LDT;
      li_Return_LDT : Int;
      lfb_TOF_Camera : TOF_TIME;
      lfb_TON_Schritt : TON_TIME;
      lfb_blinker_cam : FB_Blinker;
      lfb_blinker_config : FB_Blinker;
      lx_StartTimer : Bool;
   END_VAR



   IF lx_Init THEN


       IF gtyp_Interface_Dashboard.Subscribe.CameraPicture.ldt_ts > lldt_ts_old THEN
           lldt_ts_old := gtyp_Interface_Dashboard.Subscribe.CameraPicture.ldt_ts;
           lfb_blinker_cam(int_periodendauer := T#50ms);
       END_IF;


       QX_SSC_LED_Red_Online_Q8:= lfb_blinker_cam.outx_blinker;


       lfb_blinker_config(int_periodendauer := T#500ms);



       IF gtyp_Setup.x_Set_Pos_Activ OR gtyp_Setup.x_Color_Sensor_Calibration
                                       OR gtyp_Setup.x_Counter_Value_Calibration
                                       OR gtyp_Setup.x_Clean_Rack_HBW THEN
           QX_SSC_LED_Green_Q5  := lfb_blinker_config.outx_blinker;
           QX_SSC_LED_Yellow_Q6 := lfb_blinker_config.outx_blinker;
           QX_SSC_LED_Red_Q7    := lfb_blinker_config.outx_blinker;

       ELSIF (gtyp_Interface_Dashboard.Subscribe.State_HBW.i_code = 4)
           OR (gtyp_Interface_Dashboard.Subscribe.State_MPO.i_code = 4)
           OR (gtyp_Interface_Dashboard.Subscribe.State_SLD.i_code = 4)
           OR (gtyp_Interface_Dashboard.Subscribe.State_VGR.i_code = 4) THEN
           QX_SSC_LED_Green_Q5 := FALSE;
           QX_SSC_LED_Yellow_Q6 := FALSE;
           QX_SSC_LED_Red_Q7 := TRUE;

       ELSIF (gtyp_Interface_Dashboard.Subscribe.State_HBW.i_code = 2)
           OR (gtyp_Interface_Dashboard.Subscribe.State_MPO.i_code = 2)
           OR (gtyp_Interface_Dashboard.Subscribe.State_SLD.i_code = 2)
           OR (gtyp_Interface_Dashboard.Subscribe.State_VGR.i_code = 2) THEN
               QX_SSC_LED_Green_Q5 := FALSE;
               QX_SSC_LED_Yellow_Q6 := TRUE;
               QX_SSC_LED_Red_Q7 := FALSE;

       ELSIF (gtyp_Interface_Dashboard.Subscribe.State_HBW.i_code = 1)
           AND (gtyp_Interface_Dashboard.Subscribe.State_MPO.i_code = 1)
           AND (gtyp_Interface_Dashboard.Subscribe.State_SLD.i_code = 1)
           AND (gtyp_Interface_Dashboard.Subscribe.State_VGR.i_code = 1) THEN
               QX_SSC_LED_Green_Q5 := TRUE;
               QX_SSC_LED_Yellow_Q6 := FALSE;
               QX_SSC_LED_Red_Q7 := FALSE;

       ELSE
           QX_SSC_LED_Green_Q5 := FALSE;
           QX_SSC_LED_Yellow_Q6 := FALSE;
           QX_SSC_LED_Red_Q7 := FALSE;
       END_IF;


   ELSE
       lx_Init := TRUE;
   END_IF;
END_FUNCTION_BLOCK

FUNCTION_BLOCK PRG_DSO_Status
   VAR
      lx_Init : Bool;
      lx_Start : Bool;
      li_StepCase : Int;
      ldt_MQTT : Date_And_Time;
      li_Return_LDT : Int;
      li_code_old : Int;
      lfb_R_Trig_Outsourcing : R_TRIG;
      lfb_R_Trig_Take_Workpiece : R_TRIG;
      lfb_TON_Status : TON_TIME;
      lfb_TON_End_Order : TON_TIME;
      lx_StartStatus : Bool;
      lx_StartEndOrder : Bool;
      lx_StartTimer : Bool;
   END_VAR



   IF lx_Init THEN


       lfb_TON_Status(IN := NOT lx_StartStatus,
                       PT := T#2s);


       lfb_R_Trig_Outsourcing(CLK := NOT IX_SSC_LightBarrierOutsourcing_I4);
       lfb_R_Trig_Take_Workpiece(CLK := IX_SSC_LightBarrierOutsourcing_I4);


       IF NOT IX_SSC_LightBarrierOutsourcing_I4 AND (gtyp_Interface_Dashboard.Subscribe.State_Order.s_state = 'SHIPPED') THEN
           lx_StartEndOrder := TRUE;
       END_IF;


       lfb_TON_End_Order(IN := lx_StartEndOrder,
                          PT := T#5s);

       IF lfb_R_Trig_Take_Workpiece.Q OR lfb_TON_End_Order.Q THEN
           lx_StartEndOrder := FALSE;
           gtyp_Interface_Dashboard.Subscribe.State_Order.ldt_ts := DT_TO_LDT(ldt_MQTT);
           gtyp_Interface_Dashboard.Subscribe.State_Order.s_state := 'WAITING_FOR_ORDER';
           gtyp_Interface_Dashboard.Subscribe.State_Order.s_type := '';
           gtyp_Interface_Dashboard.Subscribe.State_DSO.x_active := FALSE;
       END_IF;


       IF (lfb_TON_Status.Q OR lfb_R_Trig_Outsourcing.Q OR lfb_R_Trig_Take_Workpiece.Q) AND NOT lx_StartStatus THEN
           lx_StartStatus := TRUE;
           li_Return_LDT := RD_SYS_T(ldt_MQTT);
           IF NOT IX_SSC_LightBarrierOutsourcing_I4 THEN
               gtyp_Interface_Dashboard.Subscribe.State_DSO.i_code := 0;
           ELSE
               gtyp_Interface_Dashboard.Subscribe.State_DSO.i_code := 1;
           END_IF;
           gtyp_Interface_Dashboard.Subscribe.State_DSO.ldt_ts := DT_TO_LDT(ldt_MQTT);
           gtyp_Interface_Dashboard.Subscribe.State_DSO.s_station := 'dso';
           gtyp_Interface_Dashboard.Subscribe.State_DSO.s_target := '';
           gtyp_Interface_Dashboard.Subscribe.State_DSO.s_description := '';
       END_IF;

       IF NOT lfb_TON_Status.Q AND lx_StartStatus THEN
           lx_StartStatus := FALSE;
       END_IF;
   ELSE
       lx_Init := TRUE;
       lx_StartEndOrder := FALSE;
   END_IF;
END_FUNCTION_BLOCK

FUNCTION_BLOCK PRG_SSC_Set_Positioning
   VAR
      lx_Init : Bool;
      lx_Start_TON_Wait : Bool;
      lx_Start_Positioning_m : Bool;
      lt_TON_Wait : Time;
      li_StepCase : Int;
      ldi_Pos_Horizontal : DInt;
      ldi_Pos_Vertical : DInt;
      lfb_R_Trig_Deaktivate : R_TRIG;
      lfb_TON_Wait : TON_TIME;
   END_VAR



   IF lx_Init THEN


       lfb_TON_Wait(IN := lx_Start_TON_Wait,
                     PT := lt_TON_Wait);

       lfb_R_Trig_Deaktivate(CLK:= NOT gtyp_Setup.x_Set_Pos_Activ
                              OR NOT ((gtyp_Setup.i_Pos_Selection > 0)
                              AND (gtyp_Setup.i_Pos_Selection < 21)));

       IF lfb_R_Trig_Deaktivate.Q THEN
           gtyp_SSC.Horizontal_Axis.x_Start_Positioning := FALSE;
           gtyp_SSC.Vertical_Axis.x_Start_Positioning := FALSE;
           gtyp_SSC.Horizontal_Axis.x_Reference := FALSE;
           gtyp_SSC.Vertical_Axis.x_Reference := FALSE;
           gtyp_Setup.x_Start_Positioning := FALSE;
           gtyp_Setup.x_Final_Positioning := FALSE;
           gtyp_Setup.x_Home_Positioning := FALSE;
           gtyp_Setup.x_Start_Offset := FALSE;
           lx_Start_Positioning_m := FALSE;
           IF (li_StepCase > 10) THEN
               li_StepCase            := 70;
           END_IF;
       END_IF;


       IF gtyp_Setup.x_Set_Pos_Activ
           AND ((gtyp_Setup.i_Pos_Selection > 0)
           AND (gtyp_Setup.i_Pos_Selection < 21))
           AND ((li_StepCase = 40)
           OR (li_StepCase = 60)) THEN



           IF gtyp_Setup.i_Pos_Selection = 1 THEN
               ldi_Pos_Horizontal := gtyp_SSC.di_Pos_Centre_Horizontal;
               ldi_Pos_Vertical := gtyp_SSC.di_Pos_Centre_Vertical;

           ELSIF gtyp_Setup.i_Pos_Selection = 2 THEN
               ldi_Pos_Horizontal := gtyp_SSC.di_Pos_HBW_Horizontal;
               ldi_Pos_Vertical := gtyp_SSC.di_Pos_HBW_Vertical;
           END_IF;
       END_IF;


       IF NOT gtyp_Setup.x_Set_Pos_Activ THEN
           gtyp_Setup.i_Pos_Selection := 0;
       END_IF;


       CASE li_StepCase OF

           0:
               lx_Start_TON_Wait := FALSE;
               li_StepCase := 10;

           10:
               IF gtyp_Setup.x_Set_Pos_Activ
                   AND ((gtyp_Setup.i_Pos_Selection > 0)
                   AND (gtyp_Setup.i_Pos_Selection < 21)) THEN
                   gtyp_SSC.Horizontal_Axis.x_Start_Positioning := FALSE;
                   gtyp_SSC.Vertical_Axis.x_Start_Positioning := FALSE;
                   gtyp_SSC.Horizontal_Axis.x_Reference := FALSE;
                   gtyp_SSC.Vertical_Axis.x_Reference := FALSE;
                   gtyp_Setup.x_Start_Positioning := FALSE;
                   gtyp_Setup.x_Final_Positioning := FALSE;
                   gtyp_Setup.x_Home_Positioning  := FALSE;
                   gtyp_Setup.x_Start_Offset := FALSE;
                   li_StepCase := 20;
               END_IF;

           20:

               gtyp_SSC.Horizontal_Axis.x_Reference := TRUE;
               gtyp_SSC.Vertical_Axis.x_Reference := TRUE;

               IF NOT gtyp_SSC.Horizontal_Axis.x_Referenced AND NOT gtyp_SSC.Vertical_Axis.x_Referenced THEN
                   li_StepCase := 30;
               END_IF;

           30:
               IF gtyp_SSC.Horizontal_Axis.x_Referenced THEN
                   gtyp_SSC.Horizontal_Axis.x_Reference := FALSE;
               END_IF;
               IF gtyp_SSC.Vertical_Axis.x_Referenced THEN
                   gtyp_SSC.Vertical_Axis.x_Reference := FALSE;
               END_IF;

               IF gtyp_SSC.Horizontal_Axis.x_Referenced AND gtyp_SSC.Vertical_Axis.x_Referenced THEN
                   gtyp_SSC.Horizontal_Axis.x_Reference := FALSE;
                   gtyp_SSC.Vertical_Axis.x_Reference := FALSE;
                   li_StepCase := 40;
               END_IF;

           40:
               IF gtyp_Setup.x_Start_Positioning OR lx_Start_Positioning_m THEN
                   lx_Start_Positioning_m := FALSE;
                   li_StepCase            := 50;
               END_IF;

           50:
               gtyp_SSC.Horizontal_Axis.di_Target_Position := ldi_Pos_Horizontal;
               gtyp_SSC.Horizontal_Axis.x_Start_Positioning := TRUE;
               gtyp_SSC.Vertical_Axis.di_Target_Position := ldi_Pos_Vertical;
               gtyp_SSC.Vertical_Axis.x_Start_Positioning := TRUE;

               IF (gtyp_SSC.Horizontal_Axis.di_Actual_Position <= (ldi_Pos_Horizontal + gtyp_SSC.Horizontal_Axis.Config.di_Pos_Window))
                   AND (gtyp_SSC.Horizontal_Axis.di_Actual_Position >= (ldi_Pos_Horizontal - gtyp_SSC.Horizontal_Axis.Config.di_Pos_Window))
                   AND gtyp_SSC.Horizontal_Axis.x_Position_Reached THEN
                   gtyp_SSC.Horizontal_Axis.x_Start_Positioning := FALSE;
               END_IF;

               IF (gtyp_SSC.Vertical_Axis.di_Actual_Position <= (ldi_Pos_Vertical + gtyp_SSC.Vertical_Axis.Config.di_Pos_Window))
                   AND (gtyp_SSC.Vertical_Axis.di_Actual_Position >= (ldi_Pos_Vertical - gtyp_SSC.Vertical_Axis.Config.di_Pos_Window))
                   AND gtyp_SSC.Vertical_Axis.x_Position_Reached THEN
                   gtyp_SSC.Vertical_Axis.x_Start_Positioning := FALSE;
               END_IF;

